(* CODESYS project 车床桁架_RECOVERED_2024-06-26T19-02-56.project
   CompiledLibraryCompatibilityVersion: LeadSysStudio V3.5 SP15 Patch 4
   Title: 车床桁架

Project tree, tasks and I/O mapping:
  Device : SC5-C0A4, Leadshine Technology Co., Ltd., order no. 504001, version 3.5.15.40
    application Application
      libraries: Standard, * (System); Util, * (System); CAA Net Base Services, 3.5.15.0 (CAA Technical Workgroup); HC_OmronUtils, 1.5.0.0 (Inovance); CmpHCUtils, 1.3.0.0 (Inovance); LS_IpoLib, 2.0.1.1 (Leadshine Technology Co.Ltd)
      task MainTask (cyclic, interval t#20ms, priority 1) calls PLC_PRG, Public_Prog, 信号, OP1002, OP1001, 回原, 气缸
      task EtherCAT_Master_Leadshine_A (cyclic, interval 4000 µs, priority 0) calls EtherCAT_Master_Leadshine_A.EtherCAT_Task, Servo_Ctrol
      program 回原 [LD]
      FunctionBlock/
        function block 点位范围判断 [ST]
        function block FB102_ClockPuls [LD]
        program Public_Prog [LD]: SystemVar
        function block FB_CylinderDouble [ST]
        function block FB_CylinderSingle [ST]
      global variables HMI
      global variables I_List
      global variables Alarm
      program POU [LD]
      Symbols
      data type CYLINDER_REF
      global variables 气缸_STRUCT
      program OP1002 [LD]: 辅助流程
      global variables System
      program 气缸 [LD]
      program Servo_Ctrol [LD]
      global variables Publics
      interface ITF
      global variables PersistentVars
      program 信号 [LD]
      program PLC_PRG [LD]
      program OP1001 [LD]
      global variables O_Lisk
    Device Diagnose
    Network Configuration
      LocalBus Config
    Resource Usage
    LocalBus_Master_Module : LocalBusR1 Master, Leadshine Technology Co., Ltd., version 3.5.15.40
      SC0032 : SC0032, Leadshine Technology Co., Ltd., version 3.5.15.40
          settings: 位置号 = 1
          unmapped channels: OUTPUT_0, OUTPUT_1, OUTPUT_2, OUTPUT_3
      SC3200 : SC3200, Leadshine Technology Co., Ltd., version 3.5.15.40
          settings: 位置号 = 0
          input  Application.I_List.X0 : BOOL  // INPUT_0.Bit0
          input  Application.I_List.X1 : BOOL  // INPUT_0.Bit1
          input  Application.I_List.X2 : BOOL  // INPUT_0.Bit2
          input  Application.I_List.X3 : BOOL  // INPUT_0.Bit3
          input  Application.I_List.X4 : BOOL  // INPUT_0.Bit4
          input  Application.I_List.X5 : BOOL  // INPUT_0.Bit5
          input  Application.I_List.X6 : BOOL  // INPUT_0.Bit6
          input  Application.I_List.X7 : BOOL  // INPUT_0.Bit7
          input  Application.I_List.X10 : BOOL  // INPUT_1.Bit0
          input  Application.I_List.X11 : BOOL  // INPUT_1.Bit1
          input  Application.I_List.X12 : BOOL  // INPUT_1.Bit2
          input  Application.I_List.X13 : BOOL  // INPUT_1.Bit3
          input  Application.I_List.X14 : BOOL  // INPUT_1.Bit4
          input  Application.I_List.X15 : BOOL  // INPUT_1.Bit5
          input  Application.I_List.X16 : BOOL  // INPUT_1.Bit6
          input  Application.I_List.X17 : BOOL  // INPUT_1.Bit7
          input  Application.I_List.X20 : BOOL  // INPUT_2.Bit0
          input  Application.I_List.X21 : BOOL  // INPUT_2.Bit1
          input  Application.I_List.X22 : BOOL  // INPUT_2.Bit2
          input  Application.I_List.X23 : BOOL  // INPUT_2.Bit3
          input  Application.I_List.X24 : BOOL  // INPUT_2.Bit4
          input  Application.I_List.X25 : BOOL  // INPUT_2.Bit5
          input  Application.I_List.X26 : BOOL  // INPUT_2.Bit6
          input  Application.I_List.X27 : BOOL  // INPUT_2.Bit7
          input  Application.I_List.X30 : BOOL  // INPUT_3.Bit0
          input  Application.I_List.X31 : BOOL  // INPUT_3.Bit1
          input  Application.I_List.X32 : BOOL  // INPUT_3.Bit2
          input  Application.I_List.X33 : BOOL  // INPUT_3.Bit3
          input  Application.I_List.X34 : BOOL  // INPUT_3.Bit4
          input  Application.I_List.X35 : BOOL  // INPUT_3.Bit5
          input  Application.I_List.X36 : BOOL  // INPUT_3.Bit6
          input  Application.I_List.X37 : BOOL  // INPUT_3.Bit7
          unmapped channels: INPUT_0, INPUT_1, INPUT_2, INPUT_3
    Modbus_Slave_RS232_COM : Modbus Slave RS232 COM, Leadshine Technology Co., Ltd., version 3.5.15.40
        settings: Vendor.Baudrate = 19200
    SoftMotion General Axis Pool
    ModbusTCP_Slave_Device : Modbus TCP Slave, Leadshine Technology Co., Ltd., version 00.00.00.10
    EtherCAT_Master_Leadshine_A : EtherCAT Master SoftMotion, 3S - Smart Software Solutions GmbH, version 3.5.16.30
        settings: NetworkName = 'ecat'; SelectNetworkByName = TRUE
      L6N_2 : L6N(COE), Leadshine Technology Co.,Ltd., order no. L6N, version Revision=16#00000001
          settings: DC sync0 cycletime = 4000; DC sync1 cycletime = 4000; Number of SDO = 6; Homing method.Index = 16#6098; Homing method.Subindex = 16#00; Homing method.Value = 19; Homing method.Size = 8; Homing method.AbortIfError = FALSE; Homing method.JumpToLine = FALSE; Homing method.Line = 0; Homing method.CompleteAccess = False; Homing velocity (fast).Index = 16#6099; Homing velocity (fast).Subindex = 16#01; Homing velocity (fast).Value = 3051735; Homing velocity (fast).Size = 32; Homing velocity (fast).AbortIfError = FALSE; Homing velocity (fast).JumpToLine = FALSE; Homing velocity (fast).Line = 0; Homing velocity (fast).CompleteAccess = False; Homing velocity (slow).Index = 16#6099; Homing velocity (slow).Subindex = 16#02; Homing velocity (slow).Value = 1220694; Homing velocity (slow).Size = 32; Homing velocity (slow).AbortIfError = FALSE; Homing velocity (slow).JumpToLine = FALSE; Homing velocity (slow).Line = 0; Homing velocity (slow).CompleteAccess = False; Homing acceleration.Index = 16#609A; Homing acceleration.Subindex = 16#00; Homing acceleration.Value = 61034692; Homing acceleration.Size = 32; Homing acceleration.AbortIfError = FALSE; Homing acceleration.JumpToLine = FALSE; Homing acceleration.Line = 0; Homing acceleration.CompleteAccess = False; Homing offset.Index = 16#607C; Homing offset.Subindex = 16#00; Homing offset.Value = 0; Homing offset.Size = 32; Homing offset.AbortIfError = FALSE;
            Homing offset.JumpToLine = FALSE; Homing offset.Line = 0; Homing offset.CompleteAccess = False
          unmapped channels: Control word, Profile target position, Touch Probe Function, Last error code, Status word, Modes of operation display, Position loop error, Actual motor torque, Actual motor position, Touch Probe Status, Touch probe pos1 pos value, Digital inputs
        Axis_2 : Axis, 3S - Smart Software Solutions GmbH, order no. 0, version 4.6.1.0
            settings: wDriveID = 2; dwRatioTechUnitsDenom = 524288000; iRatioTechUnitsNum = -859; fSWMaxVelocity = 687; fSWMaxAcceleration = 10000; fSWMaxDeceleration = 10000; fSWMaxJerk = 100000; 一圈脉冲数 = 8388608; 工作台一圈的位移 = 2; 电子齿轮比分子 = 100; 电子齿轮比分母 = 1; Commisioning.smci.Jerk = 0; ScalingIncs = 8388608; InvertDirection = True; AdrOffset_8010 = 28; BitOffset_8010 = 0; BitLength_8010 = 16; Address_8010 = '%QW14'; Type_8010 = 'UINT'; AddressPointer_8010 = ADR(%QW14); AdrOffset_8020 = 32; BitOffset_8020 = 0; BitLength_8020 = 32; Address_8020 = '%QD8'; Type_8020 = 'DINT'; AddressPointer_8020 = ADR(%QD8); AdrOffset_8030 = 4294967295; BitOffset_8030 = 0; BitLength_8030 = 32; Address_8030 = ''; Type_8030 = 'DINT'; AddressPointer_8030 = 0; AdrOffset_8040 = 4294967295; BitOffset_8040 = 0; BitLength_8040 = 16; Address_8040 = ''; Type_8040 = 'INT'; AddressPointer_8040 = 0; AdrOffset_8050 = 4294967295; BitOffset_8050 = 0;
              BitLength_8050 = 8; Address_8050 = ''; Type_8050 = 'SINT'; AddressPointer_8050 = 0; AdrOffset_8060 = 36; BitOffset_8060 = 0; BitLength_8060 = 16; Address_8060 = '%QW18'; Type_8060 = 'UINT'; AddressPointer_8060 = ADR(%QW18); AdrOffset_8070 = 4294967295; BitOffset_8070 = 0; BitLength_8070 = 0; Address_8070 = ''; Type_8070 = ''; AddressPointer_8070 = 0; AdrOffset_8080 = 4294967295; BitOffset_8080 = 0; BitLength_8080 = 16; Address_8080 = ''; Type_8080 = 'INT'; AddressPointer_8080 = 0; AdrOffset_8090 = 4294967295; BitOffset_8090 = 0; BitLength_8090 = 0; Address_8090 = ''; Type_8090 = ''; AddressPointer_8090 = 0; AdrOffset_8510 = 70; BitOffset_8510 = 0; BitLength_8510 = 16; Address_8510 = '%IW35'; Type_8510 = 'UINT'; AddressPointer_8510 = ADR(%IW35); AdrOffset_8520 = 84; BitOffset_8520 = 0; BitLength_8520 = 32; Address_8520 = '%ID21'; Type_8520 = 'DINT'; AddressPointer_8520 = ADR(%ID21);
              AdrOffset_8530 = 4294967295; BitOffset_8530 = 0; BitLength_8530 = 0; Address_8530 = ''; Type_8530 = ''; AddressPointer_8530 = 0; AdrOffset_8540 = 80; BitOffset_8540 = 0; BitLength_8540 = 16; Address_8540 = '%IW40'; Type_8540 = 'INT'; AddressPointer_8540 = ADR(%IW40); AdrOffset_8550 = 72; BitOffset_8550 = 0; BitLength_8550 = 8; Address_8550 = '%IB72'; Type_8550 = 'SINT'; AddressPointer_8550 = ADR(%IB72); AdrOffset_8560 = 96; BitOffset_8560 = 0; BitLength_8560 = 32; Address_8560 = '%ID24'; Type_8560 = 'UDINT'; AddressPointer_8560 = ADR(%ID24); AdrOffset_8570 = 88; BitOffset_8570 = 0; BitLength_8570 = 16; Address_8570 = '%IW44'; Type_8570 = 'UINT'; AddressPointer_8570 = ADR(%IW44); AdrOffset_8580 = 92; BitOffset_8580 = 0; BitLength_8580 = 32; Address_8580 = '%ID23'; Type_8580 = 'DINT'; AddressPointer_8580 = ADR(%ID23); AdrOffset_8590 = 4294967295; BitOffset_8590 = 0; BitLength_8590 = 0; Address_8590 = '';
              Type_8590 = ''; AddressPointer_8590 = 0; AdrOffset_8600 = 4294967295; BitOffset_8600 = 0; BitLength_8600 = 0; Address_8600 = ''; Type_8600 = ''; AddressPointer_8600 = 0; AdrOffset_8600 = 4294967295; BitOffset_8600 = 0; BitLength_8600 = 0; Address_8610 = ''; Type_8610 = ''; AddressPointer_8610 = 0; AdrOffset_8620 = 76; BitOffset_8620 = 0; BitLength_8620 = 32; Address_8620 = '%ID19'; Type_8620 = 'DINT'; AddressPointer_8620 = ADR(%ID19)
      L6N_1 : L6N(COE), Leadshine Technology Co.,Ltd., order no. L6N, version Revision=16#00000001
          settings: DC sync0 cycletime = 4000; DC sync1 cycletime = 4000; Number of SDO = 6; Homing method.Index = 16#6098; Homing method.Subindex = 16#00; Homing method.Value = 19; Homing method.Size = 8; Homing method.AbortIfError = FALSE; Homing method.JumpToLine = FALSE; Homing method.Line = 0; Homing method.CompleteAccess = FALSE; Homing velocity (fast).Index = 16#6099; Homing velocity (fast).Subindex = 16#01; Homing velocity (fast).Value = 8388608; Homing velocity (fast).Size = 32; Homing velocity (fast).AbortIfError = FALSE; Homing velocity (fast).JumpToLine = FALSE; Homing velocity (fast).Line = 0; Homing velocity (fast).CompleteAccess = FALSE; Homing velocity (slow).Index = 16#6099; Homing velocity (slow).Subindex = 16#02; Homing velocity (slow).Value = 3355443; Homing velocity (slow).Size = 32; Homing velocity (slow).AbortIfError = FALSE; Homing velocity (slow).JumpToLine = FALSE; Homing velocity (slow).Line = 0; Homing velocity (slow).CompleteAccess = FALSE; Homing acceleration.Index = 16#609A; Homing acceleration.Subindex = 16#00; Homing acceleration.Value = 167772160; Homing acceleration.Size = 32; Homing acceleration.AbortIfError = FALSE; Homing acceleration.JumpToLine = FALSE; Homing acceleration.Line = 0; Homing acceleration.CompleteAccess = FALSE; Homing offset.Index = 16#607C; Homing offset.Subindex = 16#00; Homing offset.Value = 0; Homing offset.Size = 32; Homing offset.AbortIfError = FALSE;
            Homing offset.JumpToLine = FALSE; Homing offset.Line = 0; Homing offset.CompleteAccess = FALSE
          unmapped channels: Control word, Profile target position, Touch Probe Function, Last error code, Status word, Modes of operation display, Position loop error, Actual motor torque, Actual motor position, Touch Probe Status, Touch probe pos1 pos value, Digital inputs
        Axis_1 : Axis, 3S - Smart Software Solutions GmbH, order no. 0, version 4.6.1.0
            settings: dwRatioTechUnitsDenom = 8388608; iRatioTechUnitsNum = -5; fSWMaxVelocity = 250; fSWMaxAcceleration = 1000; fSWMaxDeceleration = 10000; fSWMaxJerk = 100000; 一圈脉冲数 = 8388608; 工作台一圈的位移 = 5; 电子齿轮比分子 = 10; 电子齿轮比分母 = 100; ScalingIncs = 8388608; InvertDirection = True; AdrOffset_8010 = 16; BitOffset_8010 = 0; BitLength_8010 = 16; Address_8010 = '%QW8'; Type_8010 = 'UINT'; AddressPointer_8010 = ADR(%QW8); AdrOffset_8020 = 20; BitOffset_8020 = 0; BitLength_8020 = 32; Address_8020 = '%QD5'; Type_8020 = 'DINT'; AddressPointer_8020 = ADR(%QD5); AdrOffset_8030 = 4294967295; BitOffset_8030 = 0; BitLength_8030 = 32; Address_8030 = ''; Type_8030 = 'DINT'; AddressPointer_8030 = 0; AdrOffset_8040 = 4294967295; BitOffset_8040 = 0; BitLength_8040 = 16; Address_8040 = ''; Type_8040 = 'INT'; AddressPointer_8040 = 0; AdrOffset_8050 = 4294967295; BitOffset_8050 = 0; BitLength_8050 = 8; Address_8050 = '';
              Type_8050 = 'SINT'; AddressPointer_8050 = 0; AdrOffset_8060 = 24; BitOffset_8060 = 0; BitLength_8060 = 16; Address_8060 = '%QW12'; Type_8060 = 'UINT'; AddressPointer_8060 = ADR(%QW12); AdrOffset_8070 = 4294967295; BitOffset_8070 = 0; BitLength_8070 = 0; Address_8070 = ''; Type_8070 = ''; AddressPointer_8070 = 0; AdrOffset_8080 = 4294967295; BitOffset_8080 = 0; BitLength_8080 = 16; Address_8080 = ''; Type_8080 = 'INT'; AddressPointer_8080 = 0; AdrOffset_8090 = 4294967295; BitOffset_8090 = 0; BitLength_8090 = 0; Address_8090 = ''; Type_8090 = ''; AddressPointer_8090 = 0; AdrOffset_8510 = 38; BitOffset_8510 = 0; BitLength_8510 = 16; Address_8510 = '%IW19'; Type_8510 = 'UINT'; AddressPointer_8510 = ADR(%IW19); AdrOffset_8520 = 52; BitOffset_8520 = 0; BitLength_8520 = 32; Address_8520 = '%ID13'; Type_8520 = 'DINT'; AddressPointer_8520 = ADR(%ID13); AdrOffset_8530 = 4294967295; BitOffset_8530 = 0;
              BitLength_8530 = 0; Address_8530 = ''; Type_8530 = ''; AddressPointer_8530 = 0; AdrOffset_8540 = 48; BitOffset_8540 = 0; BitLength_8540 = 16; Address_8540 = '%IW24'; Type_8540 = 'INT'; AddressPointer_8540 = ADR(%IW24); AdrOffset_8550 = 40; BitOffset_8550 = 0; BitLength_8550 = 8; Address_8550 = '%IB40'; Type_8550 = 'SINT'; AddressPointer_8550 = ADR(%IB40); AdrOffset_8560 = 64; BitOffset_8560 = 0; BitLength_8560 = 32; Address_8560 = '%ID16'; Type_8560 = 'UDINT'; AddressPointer_8560 = ADR(%ID16); AdrOffset_8570 = 56; BitOffset_8570 = 0; BitLength_8570 = 16; Address_8570 = '%IW28'; Type_8570 = 'UINT'; AddressPointer_8570 = ADR(%IW28); AdrOffset_8580 = 60; BitOffset_8580 = 0; BitLength_8580 = 32; Address_8580 = '%ID15'; Type_8580 = 'DINT'; AddressPointer_8580 = ADR(%ID15); AdrOffset_8590 = 4294967295; BitOffset_8590 = 0; BitLength_8590 = 0; Address_8590 = ''; Type_8590 = ''; AddressPointer_8590 = 0;
              AdrOffset_8600 = 4294967295; BitOffset_8600 = 0; BitLength_8600 = 0; Address_8600 = ''; Type_8600 = ''; AddressPointer_8600 = 0; AdrOffset_8600 = 4294967295; BitOffset_8600 = 0; BitLength_8600 = 0; Address_8610 = ''; Type_8610 = ''; AddressPointer_8610 = 0; AdrOffset_8620 = 44; BitOffset_8620 = 0; BitLength_8620 = 32; Address_8620 = '%ID11'; Type_8620 = 'DINT'; AddressPointer_8620 = ADR(%ID11)
      L6N : L6N(COE), Leadshine Technology Co.,Ltd., order no. L6N, version Revision=16#00000001
          settings: DC sync0 cycletime = 4000; DC enable = 1; DC sync0 enable = 1; DC sync0 shift time = 0; DC sync1 cycletime = 4000; DC sync1 enable = 0; DC sync1 factor = 'x 1'; DC sync1 shift time = 0; Number of SDO = 6; Homing method.Index = 16#6098; Homing method.Subindex = 16#00; Homing method.Value = 19; Homing method.Size = 8; Homing method.AbortIfError = FALSE; Homing method.JumpToLine = FALSE; Homing method.Line = 0; Homing method.CompleteAccess = FALSE; Homing velocity (fast).Index = 16#6099; Homing velocity (fast).Subindex = 16#01; Homing velocity (fast).Value = 20971520; Homing velocity (fast).Size = 32; Homing velocity (fast).AbortIfError = FALSE; Homing velocity (fast).JumpToLine = FALSE; Homing velocity (fast).Line = 0; Homing velocity (fast).CompleteAccess = FALSE; Homing velocity (slow).Index = 16#6099; Homing velocity (slow).Subindex = 16#02; Homing velocity (slow).Value = 4194304; Homing velocity (slow).Size = 32; Homing velocity (slow).AbortIfError = FALSE; Homing velocity (slow).JumpToLine = FALSE; Homing velocity (slow).Line = 0; Homing velocity (slow).CompleteAccess = FALSE; Homing acceleration.Index = 16#609A; Homing acceleration.Subindex = 16#00; Homing acceleration.Value = 209715200; Homing acceleration.Size = 32; Homing acceleration.AbortIfError = FALSE; Homing acceleration.JumpToLine = FALSE; Homing acceleration.Line = 0;
            Homing acceleration.CompleteAccess = FALSE; Homing offset.Index = 16#607C; Homing offset.Subindex = 16#00; Homing offset.Value = 0; Homing offset.Size = 32; Homing offset.AbortIfError = FALSE; Homing offset.JumpToLine = FALSE; Homing offset.Line = 0; Homing offset.CompleteAccess = FALSE
          unmapped channels: Control word, Profile target position, Touch Probe Function, Last error code, Status word, Modes of operation display, Position loop error, Actual motor torque, Actual motor position, Touch Probe Status, Touch probe pos1 pos value, Digital inputs
        Axis : Axis, 3S - Smart Software Solutions GmbH, order no. 0, version 4.6.1.0
            settings: wDriveID = 0; dwRatioTechUnitsDenom = 2097152; iRatioTechUnitsNum = -1; fSWMaxVelocity = 200; fSWMaxAcceleration = 1000; fSWMaxDeceleration = 10000; fSWMaxJerk = 100000; 一圈脉冲数 = 10; 工作台一圈的位移 = 20; 电子齿轮比分子 = 100; 电子齿轮比分母 = 100; ScalingIncs = 8388608; InvertDirection = True; AdrOffset_8010 = 4; BitOffset_8010 = 0; BitLength_8010 = 16; Address_8010 = '%QW2'; Type_8010 = 'UINT'; AddressPointer_8010 = ADR(%QW2); AdrOffset_8020 = 8; BitOffset_8020 = 0; BitLength_8020 = 32; Address_8020 = '%QD2'; Type_8020 = 'DINT'; AddressPointer_8020 = ADR(%QD2); AdrOffset_8030 = 4294967295; BitOffset_8030 = 0; BitLength_8030 = 32; Address_8030 = ''; Type_8030 = 'DINT'; AddressPointer_8030 = 0; AdrOffset_8040 = 4294967295; BitOffset_8040 = 0; BitLength_8040 = 16; Address_8040 = ''; Type_8040 = 'INT'; AddressPointer_8040 = 0; AdrOffset_8050 = 4294967295; BitOffset_8050 = 0; BitLength_8050 = 8;
              Address_8050 = ''; Type_8050 = 'SINT'; AddressPointer_8050 = 0; AdrOffset_8060 = 12; BitOffset_8060 = 0; BitLength_8060 = 16; Address_8060 = '%QW6'; Type_8060 = 'UINT'; AddressPointer_8060 = ADR(%QW6); AdrOffset_8070 = 4294967295; BitOffset_8070 = 0; BitLength_8070 = 0; Address_8070 = ''; Type_8070 = ''; AddressPointer_8070 = 0; AdrOffset_8080 = 4294967295; BitOffset_8080 = 0; BitLength_8080 = 16; Address_8080 = ''; Type_8080 = 'INT'; AddressPointer_8080 = 0; AdrOffset_8090 = 4294967295; BitOffset_8090 = 0; BitLength_8090 = 0; Address_8090 = ''; Type_8090 = ''; AddressPointer_8090 = 0; AdrOffset_8510 = 6; BitOffset_8510 = 0; BitLength_8510 = 16; Address_8510 = '%IW3'; Type_8510 = 'UINT'; AddressPointer_8510 = ADR(%IW3); AdrOffset_8520 = 20; BitOffset_8520 = 0; BitLength_8520 = 32; Address_8520 = '%ID5'; Type_8520 = 'DINT'; AddressPointer_8520 = ADR(%ID5); AdrOffset_8530 = 4294967295;
              BitOffset_8530 = 0; BitLength_8530 = 0; Address_8530 = ''; Type_8530 = ''; AddressPointer_8530 = 0; AdrOffset_8540 = 16; BitOffset_8540 = 0; BitLength_8540 = 16; Address_8540 = '%IW8'; Type_8540 = 'INT'; AddressPointer_8540 = ADR(%IW8); AdrOffset_8550 = 8; BitOffset_8550 = 0; BitLength_8550 = 8; Address_8550 = '%IB8'; Type_8550 = 'SINT'; AddressPointer_8550 = ADR(%IB8); AdrOffset_8560 = 32; BitOffset_8560 = 0; BitLength_8560 = 32; Address_8560 = '%ID8'; Type_8560 = 'UDINT'; AddressPointer_8560 = ADR(%ID8); AdrOffset_8570 = 24; BitOffset_8570 = 0; BitLength_8570 = 16; Address_8570 = '%IW12'; Type_8570 = 'UINT'; AddressPointer_8570 = ADR(%IW12); AdrOffset_8580 = 28; BitOffset_8580 = 0; BitLength_8580 = 32; Address_8580 = '%ID7'; Type_8580 = 'DINT'; AddressPointer_8580 = ADR(%ID7); AdrOffset_8590 = 4294967295; BitOffset_8590 = 0; BitLength_8590 = 0; Address_8590 = ''; Type_8590 = '';
              AddressPointer_8590 = 0; AdrOffset_8600 = 4294967295; BitOffset_8600 = 0; BitLength_8600 = 0; Address_8600 = ''; Type_8600 = ''; AddressPointer_8600 = 0; AdrOffset_8600 = 4294967295; BitOffset_8600 = 0; BitLength_8600 = 0; Address_8610 = ''; Type_8610 = ''; AddressPointer_8610 = 0; AdrOffset_8620 = 12; BitOffset_8620 = 0; BitLength_8620 = 32; Address_8620 = '%ID3'; Type_8620 = 'DINT'; AddressPointer_8620 = ADR(%ID3)
      L6N_3 : L6N(COE), Leadshine Technology Co.,Ltd., order no. L6N, version Revision=16#00000001
          settings: DC sync0 cycletime = 4000; DC sync1 cycletime = 4000; Number of SDO = 6; Homing method.Index = 16#6098; Homing method.Subindex = 16#00; Homing method.Value = 29; Homing method.Size = 8; Homing method.AbortIfError = FALSE; Homing method.JumpToLine = FALSE; Homing method.Line = 0; Homing method.CompleteAccess = False; Homing velocity (fast).Index = 16#6099; Homing velocity (fast).Subindex = 16#01; Homing velocity (fast).Value = 3051735; Homing velocity (fast).Size = 32; Homing velocity (fast).AbortIfError = FALSE; Homing velocity (fast).JumpToLine = FALSE; Homing velocity (fast).Line = 0; Homing velocity (fast).CompleteAccess = False; Homing velocity (slow).Index = 16#6099; Homing velocity (slow).Subindex = 16#02; Homing velocity (slow).Value = 1220694; Homing velocity (slow).Size = 32; Homing velocity (slow).AbortIfError = FALSE; Homing velocity (slow).JumpToLine = FALSE; Homing velocity (slow).Line = 0; Homing velocity (slow).CompleteAccess = False; Homing acceleration.Index = 16#609A; Homing acceleration.Subindex = 16#00; Homing acceleration.Value = 61034692; Homing acceleration.Size = 32; Homing acceleration.AbortIfError = FALSE; Homing acceleration.JumpToLine = FALSE; Homing acceleration.Line = 0; Homing acceleration.CompleteAccess = False; Homing offset.Index = 16#607C; Homing offset.Subindex = 16#00; Homing offset.Value = 0; Homing offset.Size = 32; Homing offset.AbortIfError = FALSE;
            Homing offset.JumpToLine = FALSE; Homing offset.Line = 0; Homing offset.CompleteAccess = False
          unmapped channels: Control word, Profile target position, Touch Probe Function, Last error code, Status word, Modes of operation display, Position loop error, Actual motor torque, Actual motor position, Touch Probe Status, Touch probe pos1 pos value, Digital inputs
        Axis_3 : Axis, 3S - Smart Software Solutions GmbH, order no. 0, version 4.6.1.0
            settings: wDriveID = 3; dwRatioTechUnitsDenom = 3814564139; iRatioTechUnitsNum = 10000; fSWMaxVelocity = 1099; fSWMaxAcceleration = 1000; fSWMaxDeceleration = 10000; fSWMaxJerk = 100000; 一圈脉冲数 = 10; 工作台一圈的位移 = 20; 电子齿轮比分子 = 100; 电子齿轮比分母 = 100; ScalingIncs = 8388608; AdrOffset_8010 = 40; BitOffset_8010 = 0; BitLength_8010 = 16; Address_8010 = '%QW20'; Type_8010 = 'UINT'; AddressPointer_8010 = ADR(%QW20); AdrOffset_8020 = 44; BitOffset_8020 = 0; BitLength_8020 = 32; Address_8020 = '%QD11'; Type_8020 = 'DINT'; AddressPointer_8020 = ADR(%QD11); AdrOffset_8030 = 4294967295; BitOffset_8030 = 0; BitLength_8030 = 32; Address_8030 = ''; Type_8030 = 'DINT'; AddressPointer_8030 = 0; AdrOffset_8040 = 4294967295; BitOffset_8040 = 0; BitLength_8040 = 16; Address_8040 = ''; Type_8040 = 'INT'; AddressPointer_8040 = 0; AdrOffset_8050 = 4294967295; BitOffset_8050 = 0; BitLength_8050 = 8; Address_8050 = '';
              Type_8050 = 'SINT'; AddressPointer_8050 = 0; AdrOffset_8060 = 48; BitOffset_8060 = 0; BitLength_8060 = 16; Address_8060 = '%QW24'; Type_8060 = 'UINT'; AddressPointer_8060 = ADR(%QW24); AdrOffset_8070 = 4294967295; BitOffset_8070 = 0; BitLength_8070 = 0; Address_8070 = ''; Type_8070 = ''; AddressPointer_8070 = 0; AdrOffset_8080 = 4294967295; BitOffset_8080 = 0; BitLength_8080 = 16; Address_8080 = ''; Type_8080 = 'INT'; AddressPointer_8080 = 0; AdrOffset_8090 = 4294967295; BitOffset_8090 = 0; BitLength_8090 = 0; Address_8090 = ''; Type_8090 = ''; AddressPointer_8090 = 0; AdrOffset_8510 = 102; BitOffset_8510 = 0; BitLength_8510 = 16; Address_8510 = '%IW51'; Type_8510 = 'UINT'; AddressPointer_8510 = ADR(%IW51); AdrOffset_8520 = 116; BitOffset_8520 = 0; BitLength_8520 = 32; Address_8520 = '%ID29'; Type_8520 = 'DINT'; AddressPointer_8520 = ADR(%ID29); AdrOffset_8530 = 4294967295; BitOffset_8530 = 0;
              BitLength_8530 = 0; Address_8530 = ''; Type_8530 = ''; AddressPointer_8530 = 0; AdrOffset_8540 = 112; BitOffset_8540 = 0; BitLength_8540 = 16; Address_8540 = '%IW56'; Type_8540 = 'INT'; AddressPointer_8540 = ADR(%IW56); AdrOffset_8550 = 104; BitOffset_8550 = 0; BitLength_8550 = 8; Address_8550 = '%IB104'; Type_8550 = 'SINT'; AddressPointer_8550 = ADR(%IB104); AdrOffset_8560 = 128; BitOffset_8560 = 0; BitLength_8560 = 32; Address_8560 = '%ID32'; Type_8560 = 'UDINT'; AddressPointer_8560 = ADR(%ID32); AdrOffset_8570 = 120; BitOffset_8570 = 0; BitLength_8570 = 16; Address_8570 = '%IW60'; Type_8570 = 'UINT'; AddressPointer_8570 = ADR(%IW60); AdrOffset_8580 = 124; BitOffset_8580 = 0; BitLength_8580 = 32; Address_8580 = '%ID31'; Type_8580 = 'DINT'; AddressPointer_8580 = ADR(%ID31); AdrOffset_8590 = 4294967295; BitOffset_8590 = 0; BitLength_8590 = 0; Address_8590 = ''; Type_8590 = ''; AddressPointer_8590 = 0;
              AdrOffset_8600 = 4294967295; BitOffset_8600 = 0; BitLength_8600 = 0; Address_8600 = ''; Type_8600 = ''; AddressPointer_8600 = 0; AdrOffset_8600 = 4294967295; BitOffset_8600 = 0; BitLength_8600 = 0; Address_8610 = ''; Type_8610 = ''; AddressPointer_8610 = 0; AdrOffset_8620 = 108; BitOffset_8620 = 0; BitLength_8620 = 32; Address_8620 = '%ID27'; Type_8620 = 'DINT'; AddressPointer_8620 = ADR(%ID27)
*)

// Device/Application/CYLINDER_REF
TYPE CYLINDER_REF :
STRUCT
	///初始化时返回原位控制
	xInit: BOOL;
	///自动控制,变为TRUE时，执行到位控制，变为FALSE时执行原位控制
	xAutoCmd: BOOL;
	///到位标志,处于原位状态
	xIsBack: BOOL;
	///到位标志,处于到位状态	
	xIsFront: BOOL;
END_STRUCT
END_TYPE

// Device/Application/HMI
{attribute 'qualified_only'}
VAR_GLOBAL
END_VAR
VAR_GLOBAL
	报警复位 AT %MX0.0: BOOL;
END_VAR
VAR_GLOBAL RETAIN PERSISTENT
	上料推出气缸原位延时 AT %MW1002: WORD := 10;
	上料推出气缸到位延时 AT %MW1003: WORD := 10;
END_VAR
VAR_GLOBAL
	上料顶起气缸_ON_UP AT %MX0.3: BOOL;
END_VAR
VAR_GLOBAL RETAIN PERSISTENT
	上料顶起气缸原位延时 AT %MW1000: WORD := 10;
	上料顶起气缸到位位延时 AT %MW1001: WORD := 10;
END_VAR
VAR_GLOBAL
	上料气动振动筛_ON_UP AT %MX0.6: BOOL;
	X轴失能 AT %MX0.7: BOOL;
	Z2轴失能 AT %MX1.0: BOOL;
	Z1轴失能 AT %MX1.1: BOOL;
	Y轴失能 AT %MX1.2: BOOL;
	X轴_CCW AT %MX1.3: BOOL;
	X轴_CW AT %MX1.4: BOOL;
	Y轴_CCW AT %MX1.5: BOOL;
	Y轴_CW AT %MX0.5: BOOL;
	Z1轴_CCW AT %MX0.4: BOOL;
	Z1轴_CW AT %MX1.6: BOOL;
	Z2轴_CCW AT %MX0.2: BOOL;
	Z2轴_CW AT %MX0.1: BOOL;
	上料推出气缸_ON_UP AT %MX1.7: BOOL;
END_VAR
VAR_GLOBAL RETAIN PERSISTENT
	X轴手动速度 AT %MD1000: REAL := 20;
	Z1轴手动速度 AT %MD1002: REAL := 20;
	Y轴手动速度 AT %MD1001: REAL := 20;
	Z2轴手动速度 AT %MD1003: REAL := 20;
	X轴手动减速度: REAL := 1000;
	X轴手动加速度: REAL := 1000;
	Y轴手动加速度: REAL := 1000;
	Y轴手动减速度: REAL := 1000;
	Z1轴手动减速度: REAL := 1000;
	Z1轴手动加速度: REAL := 1000;
	Z2轴手动减速度: REAL := 1000;
	Z2轴手动加速度: REAL := 1000;
END_VAR
VAR_GLOBAL
	X轴错误代码 AT %MD30000: DWORD;
	X状态_未使能 AT %MX2.4: BOOL;
	X状态_报错 AT %MX2.5: BOOL;
	X状态_停止中 AT %MX2.6: BOOL;
	X状态_准备好 AT %MX2.7: BOOL;
	X状态_点位运动 AT %MX3.0: BOOL;
	X状态_连续运动: BOOL;
	X状态_同步运动: BOOL;
	X状态_回零中: BOOL;
	X状态_恒速运动 AT %MX3.1: BOOL;
	X状态_加速中 AT %MX3.2: BOOL;
	X状态_减速中 AT %MX3.3: BOOL;
	X状态_超过软限制 AT %MX3.4: BOOL;
	Y轴错误代码 AT %MD30001: DWORD;
	Y状态_未使能 AT %MX3.5: BOOL;
	Y状态_报错 AT %MX3.6: BOOL;
	Y状态_停止中 AT %MX3.7: BOOL;
	Y状态_准备好 AT %MX4.0: BOOL;
	Y状态_点位运动 AT %MX4.1: BOOL;
	Y状态_连续运动: BOOL;
	Y状态_同步运动: BOOL;
	Y状态_回零中: BOOL;
	Y状态_恒速运动 AT %MX4.2: BOOL;
	Y状态_加速中 AT %MX4.3: BOOL;
	Y状态_减速中 AT %MX4.4: BOOL;
	Y状态_超过软限制 AT %MX4.5: BOOL;
	Z1轴错误代码 AT %MD30002: DWORD;
	Z1状态_未使能 AT %MX4.6: BOOL;
	Z1状态_报错 AT %MX4.7: BOOL;
	Z1状态_停止中 AT %MX5.0: BOOL;
	Z1状态_准备好 AT %MX5.1: BOOL;
	Z1状态_点位运动 AT %MX5.2: BOOL;
	Z1状态_连续运动: BOOL;
	Z1状态_同步运动: BOOL;
	Z1状态_回零中: BOOL;
	Z1状态_恒速运动 AT %MX5.3: BOOL;
	Z1状态_加速中 AT %MX5.4: BOOL;
	Z1状态_减速中 AT %MX5.5: BOOL;
	Z1状态_超过软限制 AT %MX5.6: BOOL;
	Z2轴错误代码 AT %MD30003: DWORD;
	Z2状态_未使能 AT %MX5.7: BOOL;
	Z2状态_报错 AT %mx6.0: BOOL;
	Z2状态_停止中 AT %mx6.1: BOOL;
	Z2状态_准备好 AT %MX6.7: BOOL;
	Z2状态_点位运动 AT %MX6.2: BOOL;
	Z2状态_连续运动: BOOL;
	Z2状态_同步运动: BOOL;
	Z2状态_回零中: BOOL;
	Z2状态_恒速运动 AT %MX6.3: BOOL;
	Z2状态_加速中 AT %MX6.4: BOOL;
	Z2状态_减速中 AT %MX6.5: BOOL;
	Z2状态_超过软限制 AT %MX6.6: BOOL;
	上料气爪_ON_UP AT %MX2.3: BOOL;
	开门气缸_ON_UP AT %MX2.2: BOOL;
	翻转气缸_ON_UP AT %MX2.1: BOOL;
	下料气爪_ON_UP AT %MX2.0: BOOL;
END_VAR
VAR_GLOBAL RETAIN PERSISTENT
	点位P0 AT %MD2000: ARRAY[0..3] OF REAL;
	点位P1 AT %MD2004: ARRAY[0..3] OF REAL;
END_VAR

VAR_GLOBAL
	Y轴当前位置 AT %MD1005: REAL;
	Z2轴当前位置 AT %MD1007: REAL;
	Z1轴当前位置 AT %MD1006: REAL;
	X轴当前位置 AT %MD1004: REAL;
	Z2当前速度: REAL;
	Z1当前速度: REAL;
	Y轴当前速度: REAL;
	X轴当前速度: REAL;
END_VAR
VAR_GLOBAL RETAIN PERSISTENT
	上料气爪原位延时 AT %MW1004: WORD := 10;
	上料气爪到位延时 AT %MW1005: WORD := 10;
	下料气爪到位延时 AT %MW1006: WORD := 10;
	下料气爪原位延时 AT %MW1007: WORD := 10;
	翻转气爪到位延时 AT %MW1008: WORD := 10;
	翻转气爪原位延时 AT %MW1009: WORD := 10;
	开门气缸原位延时 AT %MW1010: WORD := 50;
	开门气缸到位延时 AT %MW1011: WORD := 50;
	点位P9 AT %MD2036: ARRAY[0..3] OF REAL;
	点位P8 AT %MD2032: ARRAY[0..3] OF REAL;
	点位P7 AT %MD2028: ARRAY[0..3] OF REAL;
	点位P6 AT %MD2024: ARRAY[0..3] OF REAL;
	点位P5 AT %MD2020: ARRAY[0..3] OF REAL;
	点位P4 AT %MD2016: ARRAY[0..3] OF REAL;
	点位P3 AT %MD2012: ARRAY[0..3] OF REAL;
	点位P2 AT %MD2008: ARRAY[0..3] OF REAL;
	点位P10 AT %MD2040: ARRAY[0..3] OF REAL;
END_VAR
VAR_GLOBAL
	Z2回零触发 AT %MX7.3: BOOL;
	Z1回零触发 AT %MX7.2: BOOL;
	Y回零触发 AT %MX7.1: BOOL;
	X回零触发 AT %MX7.0: BOOL;
	Y回零完成 AT %MX7.5: BOOL;
	Z2回零完成 AT %MX7.7: BOOL;
	Z1回零完成 AT %MX7.6: BOOL;
	X回零完成 AT %MX7.4: BOOL;
	空循环模式 AT %MX8.0: BOOL;
	排空模式 AT %MX8.1: BOOL;
	P1范围内 AT %MX8.2: BOOL;
	P2范围内 AT %MX8.3: BOOL;
	P3范围内 AT %MX8.4: BOOL;
	P4范围内 AT %MX8.5: BOOL;
	P5范围内 AT %MX8.6: BOOL;
	P6范围内 AT %MX8.7: BOOL;
	P7范围内 AT %MX9.0: BOOL;
	P8范围内 AT %MX9.1: BOOL;
	P9范围内 AT %MX9.2: BOOL;
	P10范围内 AT %MX9.3: BOOL;
END_VAR
VAR_GLOBAL RETAIN PERSISTENT
	点位P12 AT %MD2048: ARRAY[0..3] OF REAL;
	点位P11 AT %MD2044: ARRAY[0..3] OF REAL;
	点位P13 AT %MD2052: ARRAY[0..3] OF REAL;
	点位P14 AT %MD2056: ARRAY[0..3] OF REAL;
END_VAR
VAR_GLOBAL
	原点状态 AT %MW1012: WORD := 0;
	设备回原触发 AT %MX9.4: BOOL;
	设备状态 AT %MW1013: WORD;
END_VAR
VAR_GLOBAL RETAIN PERSISTENT
	X最大速度 AT %MD1010: REAL := 100;
	Y最大速度 AT %MD1011: REAL := 100;
	Z1最大速度 AT %MD1012: REAL := 100;
	Z2最大速度 AT %MD1013: REAL := 100;
	X速度比例 AT %MD1014: REAL := 10;
	Y速度比例 AT %MD1015: REAL := 10;
	Z1速度比例 AT %MD1016: REAL := 10;
	Z2速度比例 AT %MD1017: REAL := 10;
END_VAR

// Device/Application/I_List
{attribute 'qualified_only'}
VAR_GLOBAL
	// 上料传送带到位确认
	X0: BOOL;
	// 紧急停止
	X1: BOOL;
	// 推出气缸原位
	X2: BOOL;
	// 推出气缸动作位
	X3: BOOL;
	// 顶起气缸原位
	X4: BOOL;
	// 顶起气缸动作位
	X5: BOOL;
	// 上料气爪原位
	X6: BOOL;
	// 上料气爪动作位
	X7: BOOL;
	// 下料气爪原位
	X10: BOOL;
	// 下料气爪动作位
	X11: BOOL;
	// 翻转气缸原位
	X12: BOOL;
	// 翻转气缸动作位
	X13: BOOL;
	// 开门气缸原位
	X14: BOOL;
	// 开门气缸动作位
	X15: BOOL;
	// 启动按钮
	X16: BOOL;
	// 停止按钮
	X17: BOOL;
	// 复位按钮
	X20: BOOL;
	// 手自动按钮ON为自动
	X21: BOOL;
	// 下料确认
	X22: BOOL;
	// 联机卡盘夹紧
	X23: BOOL;
	// 联机启动
	X24: BOOL;
	// 联机停止
	X25: BOOL;
	// 联机故障
	X26: BOOL;
	// 联机X轴零点
	X27: BOOL;
	// 联机Z轴零点
	X30: BOOL;
	// 门
	X31: BOOL;
	// 门
	X32: BOOL;
	// 油泵报警
	X33: BOOL;
	X34: BOOL;
	X35: BOOL;
	X36: BOOL;
	X37: BOOL;
END_VAR

// Device/Application/Alarm
{attribute 'qualified_only'}
VAR_GLOBAL
END_VAR
VAR_GLOBAL
	设备急停 AT %MX100.0: BOOL;
	推出气缸手自动不一致报警 AT %MX100.1: BOOL;
	推出气缸原位报警 AT %MX100.2: BOOL;
	推出气缸到位报警 AT %MX100.3: BOOL;
	顶起气缸手自动不一致报警 AT %MX100.4: BOOL;
	顶起气缸原位报警 AT %MX100.5: BOOL;
	顶起气缸到位报警 AT %MX100.6: BOOL;
	上料气爪手自动不一致报警 AT %MX100.7: BOOL;
	上料气爪原位报警 AT %MX101.0: BOOL;
	上料气爪到位报警 AT %MX101.1: BOOL;
	下料气爪手自动不一致报警 AT %MX101.2: BOOL;
	下料气爪原位报警 AT %MX101.3: BOOL;
	下料气爪到位报警 AT %MX101.4: BOOL;
	翻转气缸手自动不一致报警 AT %MX101.5: BOOL;
	翻转气缸原位报警 AT %MX101.6: BOOL;
	翻转气缸到位报警 AT %MX101.7: BOOL;
	开门气缸手自动不一致报警 AT %MX102.0: BOOL;
	开门气缸原位报警 AT %MX102.1: BOOL;
	开门气缸到位报警 AT %MX102.2: BOOL;
END_VAR

// Device/Application/气缸_STRUCT
{attribute 'qualified_only'}
VAR_GLOBAL
	上料推出气缸: CYLINDER_REF;
	上料顶起气缸: CYLINDER_REF;
	上料振动筛: CYLINDER_REF;
	开门气缸: CYLINDER_REF;
	翻转气缸: CYLINDER_REF;
	上料气爪: CYLINDER_REF;
	下料气爪: CYLINDER_REF;
END_VAR

// Device/Application/System
{attribute 'qualified_only'}
VAR_GLOBAL
	// 上电扫描一周期
FirstScan    :BOOL;
// 常ON
AlwaysTRUE   : BOOL;
// 常OFF
AlwaysFALSE  : BOOL;
// 0.1S周期脉冲
Clock_10Hz    :BOOL;
// 0.2S周期脉冲
Clock_5Hz    :BOOL;
// 0.5S周期脉冲
Clock_2Hz    :BOOL;
// 1S周期脉冲
Clock_1Hz    :BOOL;
// 2S周期脉冲
Clock_HalfHz :BOOL;
END_VAR

// Device/Application/Publics
{attribute 'qualified_only'}
VAR_GLOBAL
	// 调试使用常ON
CYGIA_ON   :BOOL;
// 调试使用常OFF
CYGIA_OFF  :BOOL;
	启动上升: BOOL;
	警报: BOOL;
	暂停: BOOL;
	EMG: BOOL;
	X定位数据: REAL;
	Y定位数据: REAL;
	Z1定位数据: REAL;
	Z2定位数据: REAL;
END_VAR
VAR_GLOBAL RETAIN PERSISTENT
	Z2加速度 AT %MD1083: REAL;
	Z1加速度 AT %MD1082: REAL;
	Y加速度 AT %MD1081: REAL;
	X加速度 AT %MD1080: REAL;
	Z2减速度 AT %MD1087: REAL;
	Z1减速度 AT %MD1086: REAL;
	Y减速度 AT %MD1085: REAL;
	X减速度 AT %MD1084: REAL;
	Z2自动速度: REAL;
	Z1自动速度: REAL;
	Y自动速度: REAL;
	X自动速度: REAL;
END_VAR
VAR_GLOBAL
	Z2轴完成: BOOL;
	Z1轴完成: BOOL;
	Y轴完成: BOOL;
	X轴完成: BOOL;
	Z2轴启动: BOOL;
	Z1轴启动: BOOL;
	Y轴启动: BOOL;
	X轴启动: BOOL;
END_VAR

// Device/Application/PersistentVars
{attribute 'qualified_only'}
VAR_GLOBAL PERSISTENT RETAIN
	// 生成持久变量的实例路径
	HMI.上料推出气缸原位延时: WORD := WORD#10;
	// 生成持久变量的实例路径
	HMI.上料推出气缸到位延时: WORD := WORD#10;
	// 生成持久变量的实例路径
	HMI.上料顶起气缸原位延时: WORD := WORD#10;
	// 生成持久变量的实例路径
	HMI.上料顶起气缸到位位延时: WORD := WORD#10;
	// 生成持久变量的实例路径
	HMI.X轴手动速度: REAL := 20.0;
	// 生成持久变量的实例路径
	HMI.Z1轴手动速度: REAL := 20.0;
	// 生成持久变量的实例路径
	HMI.Y轴手动速度: REAL := 20.0;
	// 生成持久变量的实例路径
	HMI.Z2轴手动速度: REAL := 20.0;
	// 生成持久变量的实例路径
	HMI.X轴手动减速度: REAL := 1000.0;
	// 生成持久变量的实例路径
	HMI.X轴手动加速度: REAL := 1000.0;
	// 生成持久变量的实例路径
	HMI.Y轴手动加速度: REAL := 1000.0;
	// 生成持久变量的实例路径
	HMI.Y轴手动减速度: REAL := 1000.0;
	// 生成持久变量的实例路径
	HMI.Z1轴手动减速度: REAL := 1000.0;
	// 生成持久变量的实例路径
	HMI.Z1轴手动加速度: REAL := 1000.0;
	// 生成持久变量的实例路径
	HMI.Z2轴手动减速度: REAL := 1000.0;
	// 生成持久变量的实例路径
	HMI.Z2轴手动加速度: REAL := 1000.0;
	// 生成持久变量的实例路径
	HMI.点位P1: ARRAY [0..3] OF REAL;
	// 生成持久变量的实例路径
	HMI.点位P0: ARRAY [0..3] OF REAL;
	// 生成持久变量的实例路径
	HMI.点位P9: ARRAY [0..3] OF REAL;
	// 生成持久变量的实例路径
	HMI.点位P8: ARRAY [0..3] OF REAL;
	// 生成持久变量的实例路径
	HMI.点位P7: ARRAY [0..3] OF REAL;
	// 生成持久变量的实例路径
	HMI.点位P6: ARRAY [0..3] OF REAL;
	// 生成持久变量的实例路径
	HMI.点位P5: ARRAY [0..3] OF REAL;
	// 生成持久变量的实例路径
	HMI.点位P4: ARRAY [0..3] OF REAL;
	// 生成持久变量的实例路径
	HMI.点位P3: ARRAY [0..3] OF REAL;
	// 生成持久变量的实例路径
	HMI.点位P2: ARRAY [0..3] OF REAL;
	// 生成持久变量的实例路径
	HMI.点位P10: ARRAY [0..3] OF REAL;
	// 生成持久变量的实例路径
	HMI.上料气爪原位延时: WORD := WORD#10;
	// 生成持久变量的实例路径
	HMI.上料气爪到位延时: WORD := WORD#10;
	// 生成持久变量的实例路径
	HMI.下料气爪到位延时: WORD := WORD#10;
	// 生成持久变量的实例路径
	HMI.下料气爪原位延时: WORD := WORD#10;
	// 生成持久变量的实例路径
	HMI.翻转气爪到位延时: WORD := WORD#10;
	// 生成持久变量的实例路径
	HMI.翻转气爪原位延时: WORD := WORD#10;
	// 生成持久变量的实例路径
	HMI.开门气缸原位延时: WORD := 50;
	// 生成持久变量的实例路径
	HMI.开门气缸到位延时: WORD := 50;
	// 生成持久变量的实例路径
	Publics.Y加速度: REAL;
	// 生成持久变量的实例路径
	Publics.X加速度: REAL;
	// 生成持久变量的实例路径
	Publics.Z2减速度: REAL;
	// 生成持久变量的实例路径
	Publics.Z1减速度: REAL;
	// 生成持久变量的实例路径
	Publics.Y减速度: REAL;
	// 生成持久变量的实例路径
	Publics.X减速度: REAL;
	// 生成持久变量的实例路径
	Publics.Z2自动速度: REAL;
	// 生成持久变量的实例路径
	Publics.Z1自动速度: REAL;
	// 生成持久变量的实例路径
	Publics.Y自动速度: REAL;
	// 生成持久变量的实例路径
	Publics.X自动速度: REAL;
	// 生成持久变量的实例路径
	HMI.点位P12: ARRAY [0..3] OF REAL;
	// 生成持久变量的实例路径
	HMI.点位P11: ARRAY [0..3] OF REAL;
	// 生成持久变量的实例路径
	HMI.点位P13: ARRAY [0..3] OF REAL;
	// 生成持久变量的实例路径
	HMI.点位P14: ARRAY [0..3] OF REAL;
	// 生成持久变量的实例路径
	HMI.X最大速度: REAL := 100.0;
	// 生成持久变量的实例路径
	HMI.Y最大速度: REAL := 100.0;
	// 生成持久变量的实例路径
	HMI.Z1最大速度: REAL := 100.0;
	// 生成持久变量的实例路径
	HMI.Z2最大速度: REAL := 100.0;
	// 生成持久变量的实例路径
	HMI.X速度比例: REAL := 10.0;
	// 生成持久变量的实例路径
	HMI.Y速度比例: REAL := 10.0;
	// 生成持久变量的实例路径
	HMI.Z1速度比例: REAL := 10.0;
	// 生成持久变量的实例路径
	HMI.Z2速度比例: REAL := 10.0;
	// 生成持久变量的实例路径
	Publics.Z2加速度: REAL;
	// 生成持久变量的实例路径
	Publics.Z1加速度: REAL;
END_VAR

// Device/Application/O_Lisk
{attribute 'qualified_only'}
VAR_GLOBAL
	// 皮带运转
	Y0 AT %QX0.0: BOOL;
	// 震动筛运动
	Y1 AT %QX0.1: BOOL;
	// 推出气缸原位
	Y2 AT %QX0.2: BOOL;
	// 紧急停止输出
	Y3 AT %QX0.3: BOOL;
	// 顶起气缸原位
	Y4 AT %QX0.4: BOOL;
	Y5 AT %QX0.5: BOOL;
	// 上料气爪原位
	Y6 AT %QX0.6: BOOL;
	Y7 AT %QX0.7: BOOL;
	// 下料气爪原位
	Y10 AT %QX1.0: BOOL;
	Y11 AT %QX1.1: BOOL;
	// 翻转气缸原位
	Y12 AT %QX1.2: BOOL;
	Y13 AT %QX1.3: BOOL;
	// 开门气缸原位
	Y14 AT %QX1.4: BOOL;
	Y15 AT %QX1.5: BOOL;
	// 启动按钮LED
	Y16 AT %QX1.6: BOOL;
	// 停止按钮LED
	Y17 AT %QX1.7: BOOL;
	// 复位按钮LED
	Y20 AT %QX2.0: BOOL;
	Y21 AT %QX2.1: BOOL;
	// 下料传送带
	Y22 AT %QX2.2: BOOL;
	// 三色灯红
	Y23 AT %QX2.3: BOOL;
	// 三色灯黄
	Y24 AT %QX2.4: BOOL;
	// 三色灯绿
	Y25 AT %QX2.5: BOOL;
	// 三色灯蜂鸣
	Y26 AT %QX2.6: BOOL;
	// 联机卡盘夹紧
	Y27 AT %QX2.7: BOOL;
	// 联机启动
	Y30 AT %QX3.0: BOOL;
	// 联机停止
	Y31 AT %QX3.1: BOOL;
	Y32 AT %QX3.2: BOOL;
	Y33 AT %QX3.3: BOOL;
	Y34 AT %QX3.4: BOOL;
	Y35 AT %QX3.5: BOOL;
	Y36 AT %QX3.6: BOOL;
	Y37 AT %QX3.7: BOOL;
END_VAR

// Device/Application/PLC_PRG
PROGRAM PLC_PRG

END_PROGRAM

// Device/Application/FunctionBlock/Public_Prog
PROGRAM Public_Prog
VAR
	Clock_10Hz: FB102_ClockPuls;
	Clock_5Hz: FB102_ClockPuls;
	Clock_2Hz: FB102_ClockPuls;
	Clock_1Hz: FB102_ClockPuls;
	Clock_HalfHz: FB102_ClockPuls;
END_VAR
VAR // added by the converter: edge detectors and wires of the graphical bodies
    _rt1 : R_TRIG;
END_VAR

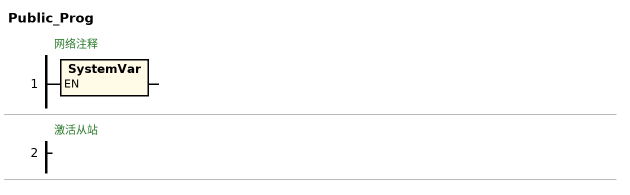
// NETWORK 1
// 网络注释
SystemVar();

// NETWORK 2
// 激活从站

ACTION SystemVar:
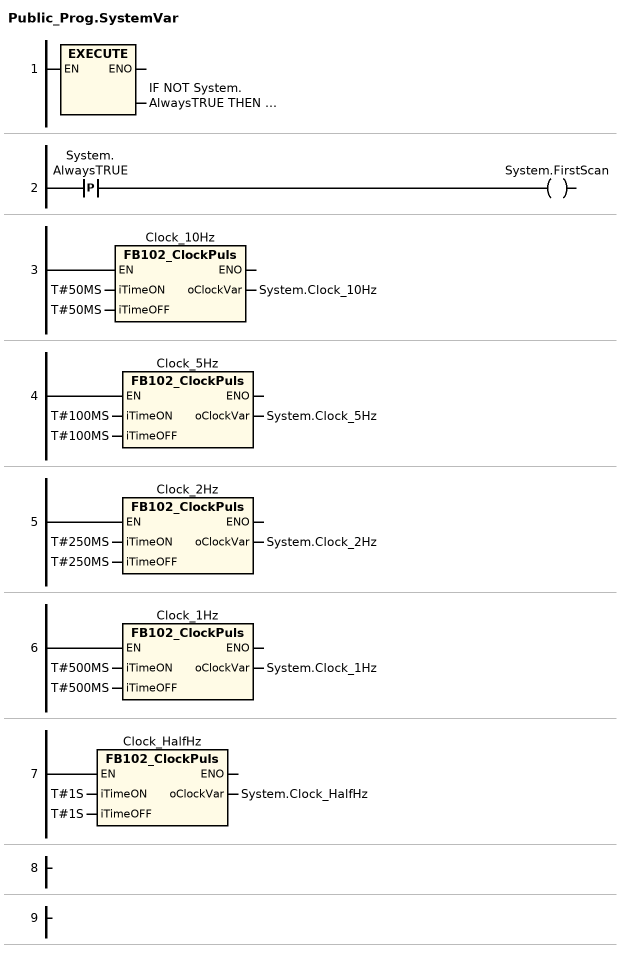
// NETWORK 1
IF NOT System.AlwaysTRUE THEN
	System.AlwaysTRUE := TRUE;
END_IF
IF  System.AlwaysFALSE THEN
	System.AlwaysFALSE := FALSE;
END_IF
IF NOT Publics.CYGIA_ON THEN
	Publics.CYGIA_ON := TRUE;
END_IF
IF  Publics.CYGIA_OFF THEN
	Publics.CYGIA_OFF := FALSE;
END_IF

// NETWORK 2
_rt1(CLK := System.AlwaysTRUE);
System.FirstScan := _rt1.Q;

// NETWORK 3
Clock_10Hz(iTimeON := T#50MS, iTimeOFF := T#50MS, oClockVar => System.Clock_10Hz); // FB102_ClockPuls

// NETWORK 4
Clock_5Hz(iTimeON := T#100MS, iTimeOFF := T#100MS, oClockVar => System.Clock_5Hz); // FB102_ClockPuls

// NETWORK 5
Clock_2Hz(iTimeON := T#250MS, iTimeOFF := T#250MS, oClockVar => System.Clock_2Hz); // FB102_ClockPuls

// NETWORK 6
Clock_1Hz(iTimeON := T#500MS, iTimeOFF := T#500MS, oClockVar => System.Clock_1Hz); // FB102_ClockPuls

// NETWORK 7
Clock_HalfHz(iTimeON := T#1S, iTimeOFF := T#1S, oClockVar => System.Clock_HalfHz); // FB102_ClockPuls

// NETWORK 8

// NETWORK 9
END_ACTION

END_PROGRAM

// Device/Application/FunctionBlock/FB102_ClockPuls
FUNCTION_BLOCK FB102_ClockPuls
VAR_INPUT
	///脉冲ON时间
	iTimeON: TIME;
	///脉冲OFF时间
	iTimeOFF: TIME;
END_VAR
VAR_OUTPUT
	///时钟脉冲差速器
	oClockVar: BOOL;
END_VAR
VAR
	TON_Clock: TON;
	TOF_Clock: TOF;
END_VAR

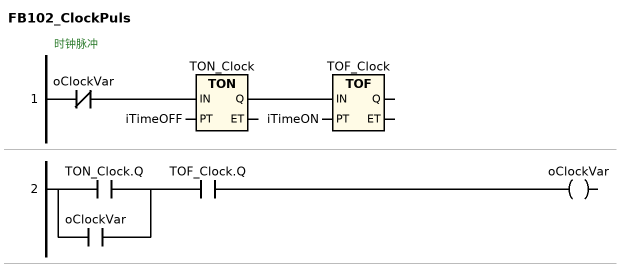
// NETWORK 1
// 时钟脉冲
TON_Clock(IN := NOT oClockVar, PT := iTimeOFF); // TON
TOF_Clock(IN := TON_Clock.Q, PT := iTimeON); // TOF

// NETWORK 2
oClockVar := (TON_Clock.Q OR oClockVar) AND TOF_Clock.Q;

END_FUNCTION_BLOCK

// Device/Application/信号
PROGRAM 信号
VAR
	循环时间传递: BOOL;
	循环时间: WORD;
	P2_Y下极限: REAL;
	P2_Y上极限: REAL;
	P2_X下极限: REAL;
	P2_X上极限: REAL;
	允许自动运行: BOOL;
	P2_Z1上极限: REAL;
	P2_Z1下极限: REAL;
	P2_Z2上极限: REAL;
	P2_Z2下极限: REAL;
	P2范围内: BOOL;
	TON_0: TON;
	循环停止通知: BOOL;
	P1: 点位范围判断;
	点位范围判断_0: 点位范围判断;
	点位范围判断_1: 点位范围判断;
	点位范围判断_2: 点位范围判断;
	点位范围判断_3: 点位范围判断;
	点位范围判断_4: 点位范围判断;
	点位范围判断_5: 点位范围判断;
	点位范围判断_6: 点位范围判断;
	点位范围判断_7: 点位范围判断;
	BLINK_0: BLINK;
	上次循环时间: WORD;
END_VAR
VAR // added by the converter: edge detectors and wires of the graphical bodies
    _w1 : BOOL;
    _rt1, _rt2 : R_TRIG;
END_VAR

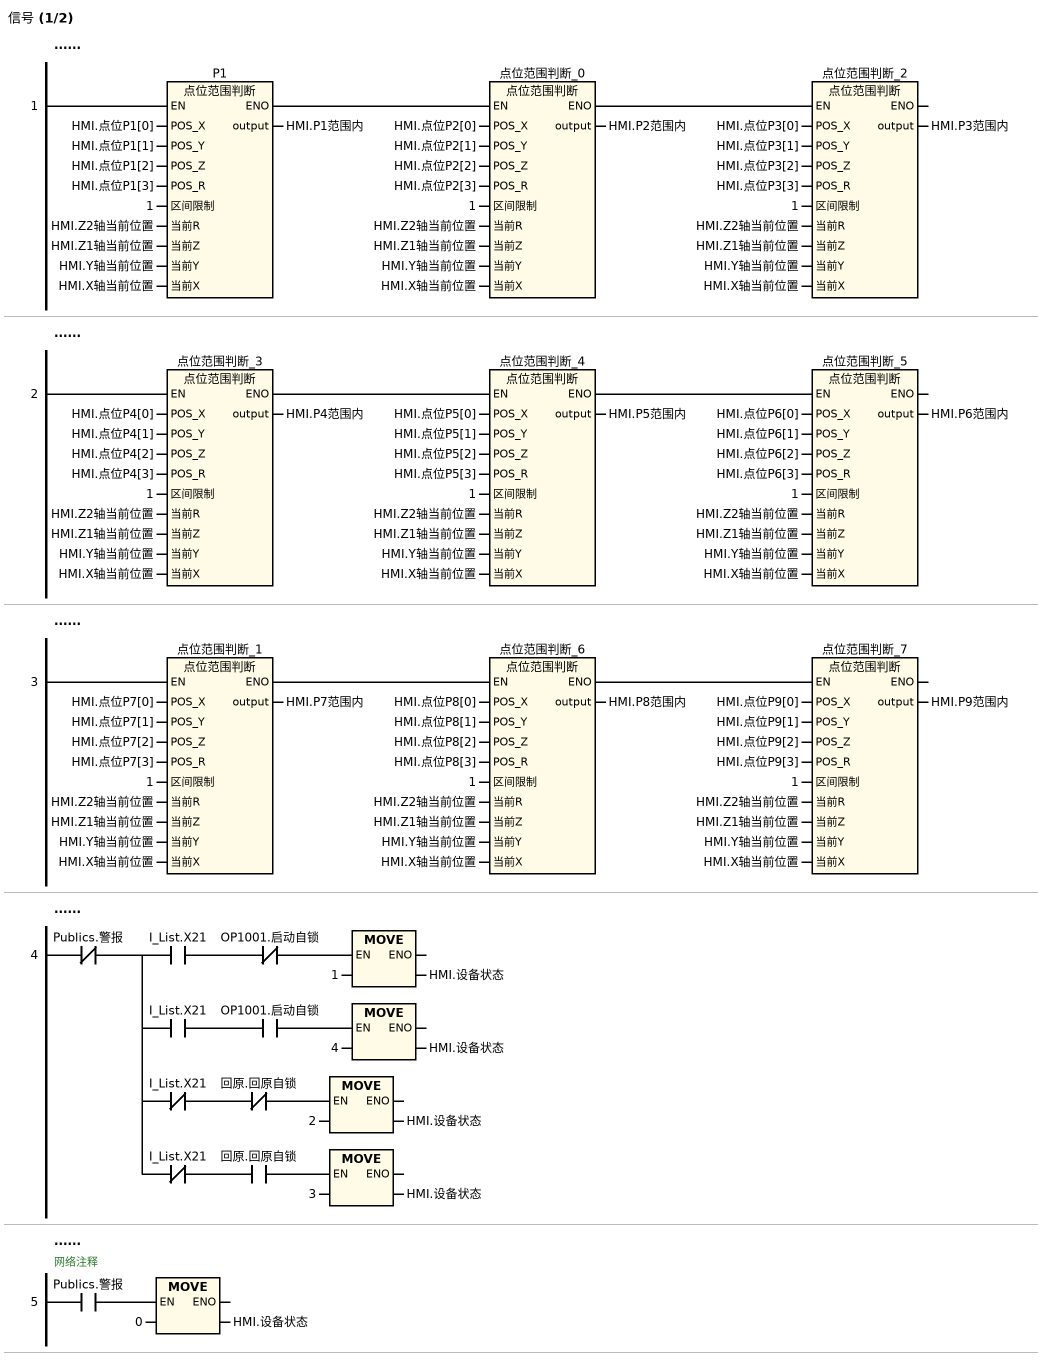
// NETWORK 1: ......
P1(
    POS_X := HMI.点位P1[0],
    POS_Y := HMI.点位P1[1],
    POS_Z := HMI.点位P1[2],
    POS_R := HMI.点位P1[3],
    区间限制 := 1,
    当前R := HMI.Z2轴当前位置,
    当前Z := HMI.Z1轴当前位置,
    当前Y := HMI.Y轴当前位置,
    当前X := HMI.X轴当前位置,
    output => HMI.P1范围内); // 点位范围判断
点位范围判断_0(
    POS_X := HMI.点位P2[0],
    POS_Y := HMI.点位P2[1],
    POS_Z := HMI.点位P2[2],
    POS_R := HMI.点位P2[3],
    区间限制 := 1,
    当前R := HMI.Z2轴当前位置,
    当前Z := HMI.Z1轴当前位置,
    当前Y := HMI.Y轴当前位置,
    当前X := HMI.X轴当前位置,
    output => HMI.P2范围内); // 点位范围判断
点位范围判断_2(
    POS_X := HMI.点位P3[0],
    POS_Y := HMI.点位P3[1],
    POS_Z := HMI.点位P3[2],
    POS_R := HMI.点位P3[3],
    区间限制 := 1,
    当前R := HMI.Z2轴当前位置,
    当前Z := HMI.Z1轴当前位置,
    当前Y := HMI.Y轴当前位置,
    当前X := HMI.X轴当前位置,
    output => HMI.P3范围内); // 点位范围判断

// NETWORK 2: ......
点位范围判断_3(
    POS_X := HMI.点位P4[0],
    POS_Y := HMI.点位P4[1],
    POS_Z := HMI.点位P4[2],
    POS_R := HMI.点位P4[3],
    区间限制 := 1,
    当前R := HMI.Z2轴当前位置,
    当前Z := HMI.Z1轴当前位置,
    当前Y := HMI.Y轴当前位置,
    当前X := HMI.X轴当前位置,
    output => HMI.P4范围内); // 点位范围判断
点位范围判断_4(
    POS_X := HMI.点位P5[0],
    POS_Y := HMI.点位P5[1],
    POS_Z := HMI.点位P5[2],
    POS_R := HMI.点位P5[3],
    区间限制 := 1,
    当前R := HMI.Z2轴当前位置,
    当前Z := HMI.Z1轴当前位置,
    当前Y := HMI.Y轴当前位置,
    当前X := HMI.X轴当前位置,
    output => HMI.P5范围内); // 点位范围判断
点位范围判断_5(
    POS_X := HMI.点位P6[0],
    POS_Y := HMI.点位P6[1],
    POS_Z := HMI.点位P6[2],
    POS_R := HMI.点位P6[3],
    区间限制 := 1,
    当前R := HMI.Z2轴当前位置,
    当前Z := HMI.Z1轴当前位置,
    当前Y := HMI.Y轴当前位置,
    当前X := HMI.X轴当前位置,
    output => HMI.P6范围内); // 点位范围判断

// NETWORK 3: ......
点位范围判断_1(
    POS_X := HMI.点位P7[0],
    POS_Y := HMI.点位P7[1],
    POS_Z := HMI.点位P7[2],
    POS_R := HMI.点位P7[3],
    区间限制 := 1,
    当前R := HMI.Z2轴当前位置,
    当前Z := HMI.Z1轴当前位置,
    当前Y := HMI.Y轴当前位置,
    当前X := HMI.X轴当前位置,
    output => HMI.P7范围内); // 点位范围判断
点位范围判断_6(
    POS_X := HMI.点位P8[0],
    POS_Y := HMI.点位P8[1],
    POS_Z := HMI.点位P8[2],
    POS_R := HMI.点位P8[3],
    区间限制 := 1,
    当前R := HMI.Z2轴当前位置,
    当前Z := HMI.Z1轴当前位置,
    当前Y := HMI.Y轴当前位置,
    当前X := HMI.X轴当前位置,
    output => HMI.P8范围内); // 点位范围判断
点位范围判断_7(
    POS_X := HMI.点位P9[0],
    POS_Y := HMI.点位P9[1],
    POS_Z := HMI.点位P9[2],
    POS_R := HMI.点位P9[3],
    区间限制 := 1,
    当前R := HMI.Z2轴当前位置,
    当前Z := HMI.Z1轴当前位置,
    当前Y := HMI.Y轴当前位置,
    当前X := HMI.X轴当前位置,
    output => HMI.P9范围内); // 点位范围判断

// NETWORK 4: ......
_w1 := NOT Publics.警报;
IF _w1 AND I_List.X21 AND NOT OP1001.启动自锁 THEN HMI.设备状态 := 1; END_IF
IF _w1 AND I_List.X21 AND OP1001.启动自锁 THEN HMI.设备状态 := 4; END_IF
IF _w1 AND NOT I_List.X21 AND NOT 回原.回原自锁 THEN HMI.设备状态 := 2; END_IF
IF _w1 AND NOT I_List.X21 AND 回原.回原自锁 THEN HMI.设备状态 := 3; END_IF

// NETWORK 5: ......
// 网络注释
IF Publics.警报 THEN HMI.设备状态 := 0; END_IF

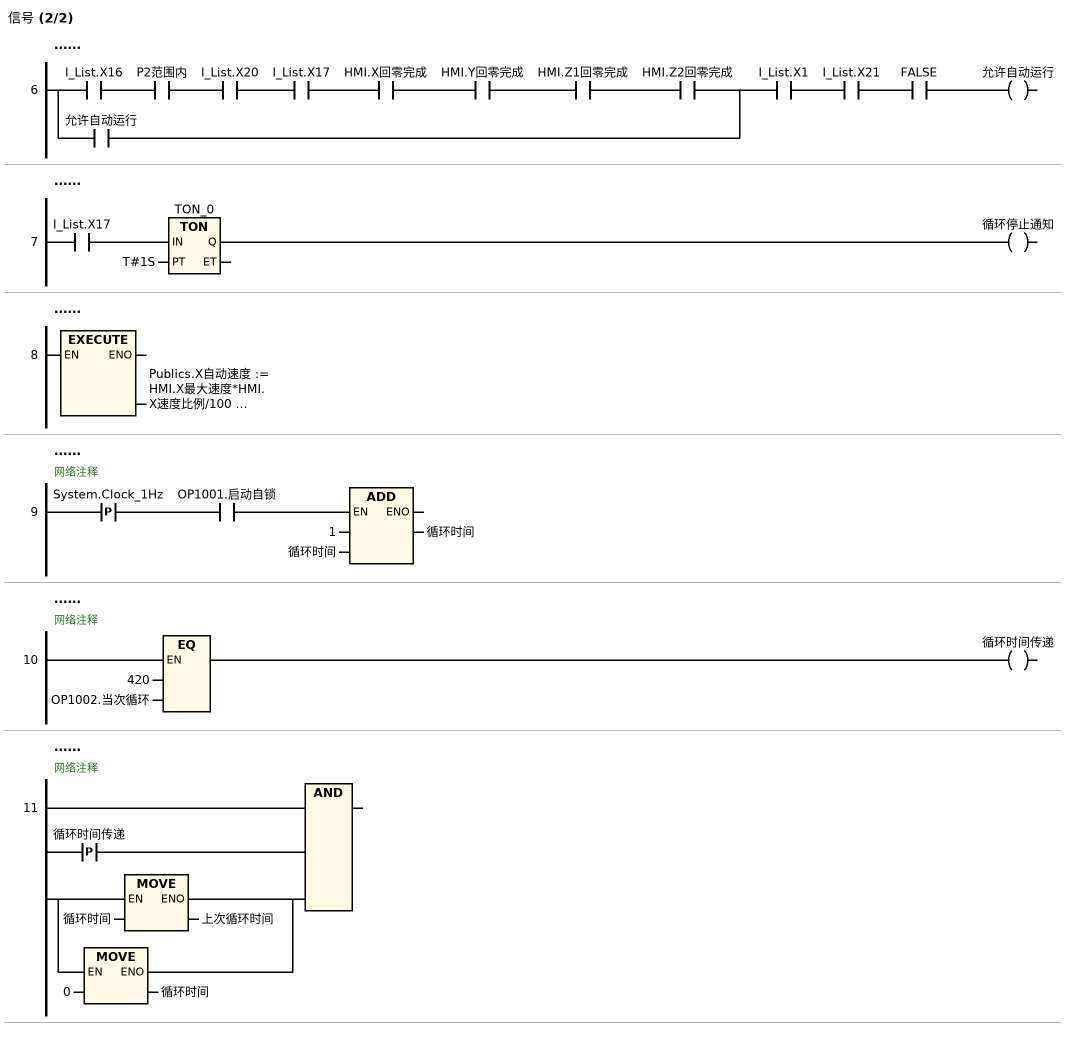
// NETWORK 6: ......
允许自动运行 := (I_List.X16 AND P2范围内 AND I_List.X20 AND I_List.X17 AND HMI.X回零完成 AND HMI.Y回零完成 AND HMI.Z1回零完成 AND HMI.Z2回零完成 OR 允许自动运行) AND I_List.X1 AND I_List.X21 AND FALSE;

// NETWORK 7: ......
TON_0(IN := I_List.X17, PT := T#1S); // TON
循环停止通知 := TON_0.Q;

// NETWORK 8: ......
Publics.X自动速度 := HMI.X最大速度*HMI.X速度比例/100;
Publics.Y自动速度 := HMI.Y最大速度*HMI.Y速度比例/100;
Publics.Z1自动速度 := HMI.Z1最大速度*HMI.Z1速度比例/100;
Publics.Z2自动速度 := HMI.Z2最大速度*HMI.Z2速度比例/100;

// NETWORK 9: ......
// 网络注释
_rt1(CLK := System.Clock_1Hz);
IF _rt1.Q AND OP1001.启动自锁 THEN 循环时间 := 1 + 循环时间; END_IF

// NETWORK 10: ......
// 网络注释
循环时间传递 := 420 = OP1002.当次循环;

// NETWORK 11: ......
// 网络注释
_rt2(CLK := 循环时间传递);
上次循环时间 := 循环时间;
循环时间 := 0;
(* _rt2.Q AND (TRUE OR TRUE); result not used *)

END_PROGRAM

// Device/Application/FunctionBlock/点位范围判断
FUNCTION_BLOCK 点位范围判断
VAR_INPUT
	POS_X: REAL;
	POS_Y: REAL;
	POS_Z: REAL;
	POS_R: REAL;
END_VAR
VAR
	X上极限: REAL;
	X下极限: REAL;
	Y上极限: REAL;
	Y下极限: REAL;
	R上极限: REAL;
	R下极限: REAL;
	Z上极限: REAL;
	Z下极限: REAL;
END_VAR
VAR_OUTPUT
	output: BOOL;
END_VAR
VAR_INPUT
	区间限制: REAL;
	当前R: REAL;
	当前Z: REAL;
	当前Y: REAL;
	当前X: REAL;
END_VAR

X上极限:=POS_X+区间限制;
X下极限:=POS_X-区间限制;
Y上极限:=POS_Y+区间限制;
Y下极限:=POS_Y-区间限制;
R上极限:=POS_Z+区间限制;
R下极限:=POS_Z-区间限制;
Z上极限:=POS_R+区间限制;
Z下极限:=POS_R-区间限制;
IF X上极限>当前X THEN
    IF X下极限<当前X THEN
		IF Y上极限>当前Y THEN
			IF Y下极限<当前Y THEN
				IF R上极限>当前R THEN
					IF R下极限<当前R THEN
						IF Z上极限>当前Z THEN
							IF Z下极限<当前Z THEN
								output:=1;	
							ELSE
								output:=0;		
							END_IF
						ELSE
							output:=0;	
						END_IF
					ELSE
						output:=0;	
					END_IF
				ELSE
					output:=0;
				END_IF
			ELSE
				output:=0;
			END_IF
		ELSE
			output:=0;
		END_IF
	ELSE
		output:=0;
	END_IF
ELSE
	output:=0;
END_IF

END_FUNCTION_BLOCK

// Device/Application/OP1001
PROGRAM OP1001
VAR
	启动自锁: BOOL;
	下次循环: word;
	当次循环: word;
	循环停止: BOOL;
	阻止运行条件: BOOL;
	TON_0: TON;
	TON_1: TON;
	TON_2: TON;
	通知_允许抓取物料: BOOL;
	A1: BOOL;
	A2: BOOL;
	A3: BOOL;
	A4: BOOL;
	A5: BOOL;
	A6: BOOL;
	A7: BOOL;
	A8: BOOL;
	启动条件: BOOL;
	DEBUG: BOOL;
END_VAR
VAR_INPUT
	通知_物料抓取完成: BOOL;
END_VAR
VAR
	流程结束: BOOL;
END_VAR
VAR // added by the converter: edge detectors and wires of the graphical bodies
    _w1, _w2, _w3, _w4, _w5, _w6, _w7, _w8 : BOOL;
    _rt1, _rt2 : R_TRIG;
END_VAR

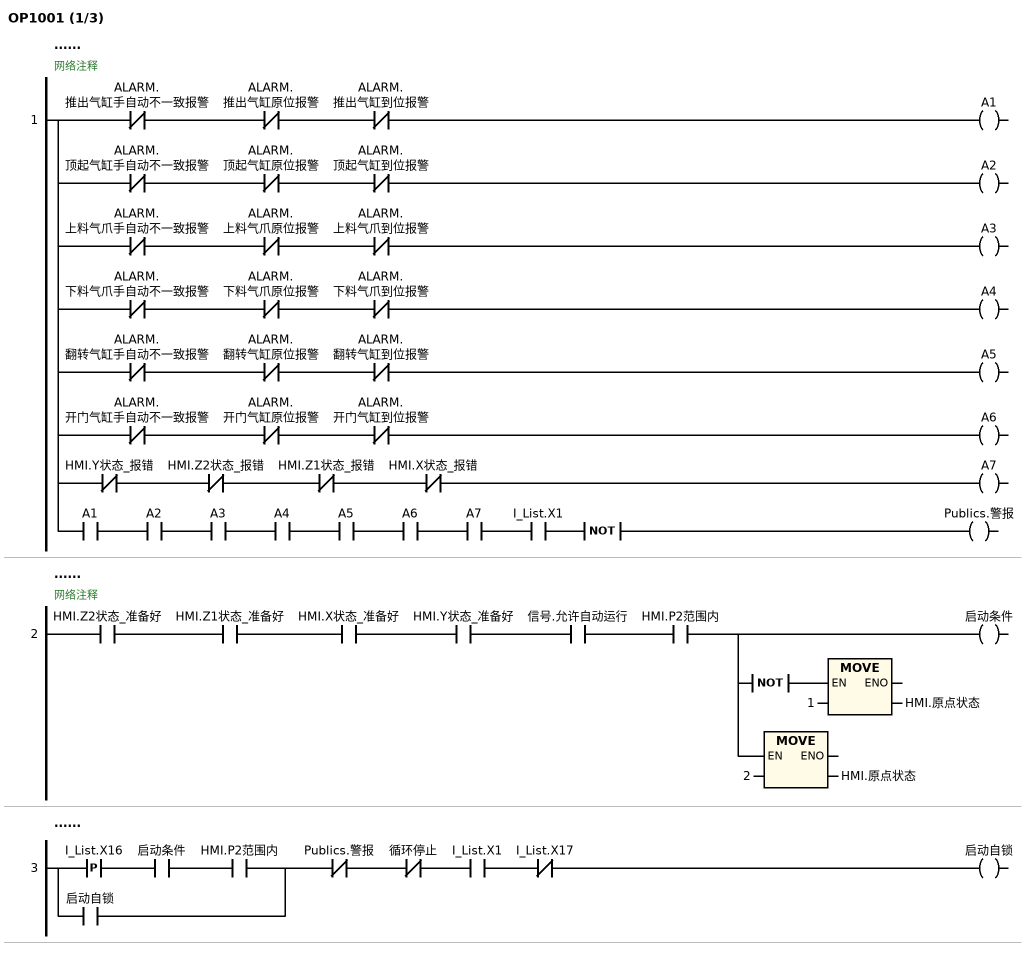
// NETWORK 1: ......
// 网络注释
A1 := NOT ALARM.推出气缸手自动不一致报警 AND NOT ALARM.推出气缸原位报警 AND NOT ALARM.推出气缸到位报警;
A2 := NOT ALARM.顶起气缸手自动不一致报警 AND NOT ALARM.顶起气缸原位报警 AND NOT ALARM.顶起气缸到位报警;
A3 := NOT ALARM.上料气爪手自动不一致报警 AND NOT ALARM.上料气爪原位报警 AND NOT ALARM.上料气爪到位报警;
A4 := NOT ALARM.下料气爪手自动不一致报警 AND NOT ALARM.下料气爪原位报警 AND NOT ALARM.下料气爪到位报警;
A5 := NOT ALARM.翻转气缸手自动不一致报警 AND NOT ALARM.翻转气缸原位报警 AND NOT ALARM.翻转气缸到位报警;
A6 := NOT ALARM.开门气缸手自动不一致报警 AND NOT ALARM.开门气缸原位报警 AND NOT ALARM.开门气缸到位报警;
A7 := NOT HMI.Y状态_报错 AND NOT HMI.Z2状态_报错 AND NOT HMI.Z1状态_报错 AND NOT HMI.X状态_报错;
Publics.警报 := NOT (A1 AND A2 AND A3 AND A4 AND A5 AND A6 AND A7 AND I_List.X1);

// NETWORK 2: ......
// 网络注释
_w1 := HMI.Z2状态_准备好 AND HMI.Z1状态_准备好 AND HMI.X状态_准备好 AND HMI.Y状态_准备好 AND 信号.允许自动运行 AND HMI.P2范围内;
启动条件 := _w1;
IF NOT _w1 THEN HMI.原点状态 := 1; END_IF
IF _w1 THEN HMI.原点状态 := 2; END_IF

// NETWORK 3: ......
_rt1(CLK := I_List.X16);
启动自锁 := (_rt1.Q AND 启动条件 AND HMI.P2范围内 OR 启动自锁) AND NOT Publics.警报 AND NOT 循环停止 AND I_List.X1 AND NOT I_List.X17;

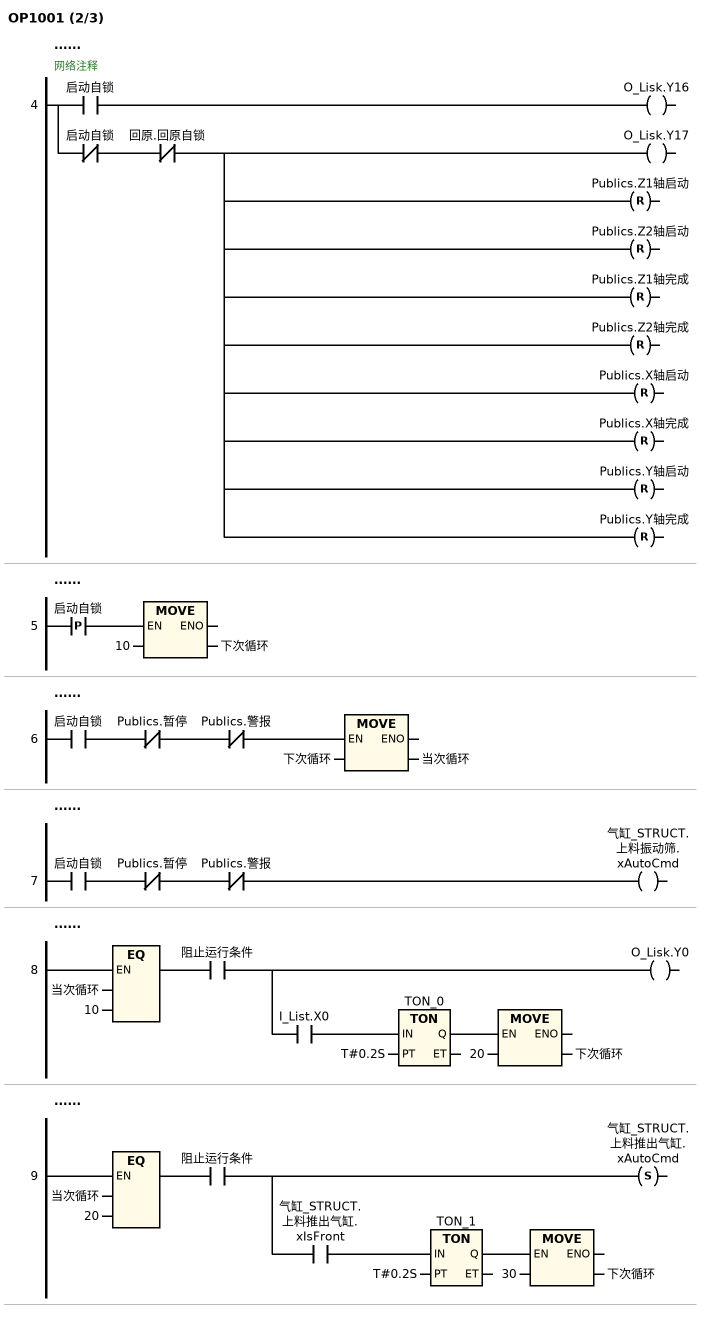
// NETWORK 4: ......
// 网络注释
O_Lisk.Y16 := 启动自锁;
_w2 := NOT 启动自锁 AND NOT 回原.回原自锁;
O_Lisk.Y17 := _w2;
Publics.Z1轴启动 R= _w2;
Publics.Z2轴启动 R= _w2;
Publics.Z1轴完成 R= _w2;
Publics.Z2轴完成 R= _w2;
Publics.X轴启动 R= _w2;
Publics.X轴完成 R= _w2;
Publics.Y轴启动 R= _w2;
Publics.Y轴完成 R= _w2;

// NETWORK 5: ......
_rt2(CLK := 启动自锁);
IF _rt2.Q THEN 下次循环 := 10; END_IF

// NETWORK 6: ......
IF 启动自锁 AND NOT Publics.暂停 AND NOT Publics.警报 THEN 当次循环 := 下次循环; END_IF

// NETWORK 7: ......
气缸_STRUCT.上料振动筛.xAutoCmd := 启动自锁 AND NOT Publics.暂停 AND NOT Publics.警报;

// NETWORK 8: ......
_w3 := 当次循环 = 10 AND 阻止运行条件;
O_Lisk.Y0 := _w3;
TON_0(IN := _w3 AND I_List.X0, PT := T#0.2S); // TON
IF TON_0.Q THEN 下次循环 := 20; END_IF

// NETWORK 9: ......
_w4 := 当次循环 = 20 AND 阻止运行条件;
气缸_STRUCT.上料推出气缸.xAutoCmd S= _w4;
TON_1(IN := _w4 AND 气缸_STRUCT.上料推出气缸.xIsFront, PT := T#0.2S); // TON
IF TON_1.Q THEN 下次循环 := 30; END_IF

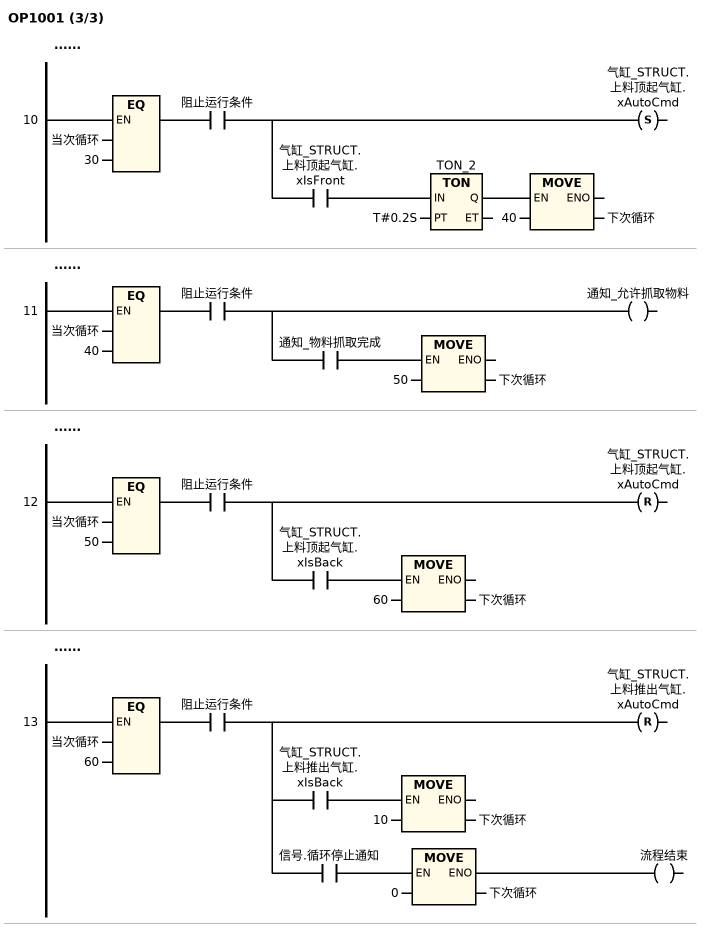
// NETWORK 10: ......
_w5 := 当次循环 = 30 AND 阻止运行条件;
气缸_STRUCT.上料顶起气缸.xAutoCmd S= _w5;
TON_2(IN := _w5 AND 气缸_STRUCT.上料顶起气缸.xIsFront, PT := T#0.2S); // TON
IF TON_2.Q THEN 下次循环 := 40; END_IF

// NETWORK 11: ......
_w6 := 当次循环 = 40 AND 阻止运行条件;
通知_允许抓取物料 := _w6;
IF _w6 AND 通知_物料抓取完成 THEN 下次循环 := 50; END_IF

// NETWORK 12: ......
_w7 := 当次循环 = 50 AND 阻止运行条件;
气缸_STRUCT.上料顶起气缸.xAutoCmd R= _w7;
IF _w7 AND 气缸_STRUCT.上料顶起气缸.xIsBack THEN 下次循环 := 60; END_IF

// NETWORK 13: ......
_w8 := 当次循环 = 60 AND 阻止运行条件;
气缸_STRUCT.上料推出气缸.xAutoCmd R= _w8;
IF _w8 AND 气缸_STRUCT.上料推出气缸.xIsBack THEN 下次循环 := 10; END_IF
IF _w8 AND 信号.循环停止通知 THEN 下次循环 := 0; END_IF
流程结束 := _w8 AND 信号.循环停止通知;

END_PROGRAM

// Device/Application/回原
PROGRAM 回原
VAR
	下次循环: WORD;
	回原条件: BOOL;
	阻止条件: BOOL;
	回原自锁: BOOL;
	当次循环: WORD;
	判断下极限: REAL;
	判断上极限: REAL;
	避开扫描周期: BOOL;
	流程结束: BOOL;
END_VAR
VAR // added by the converter: edge detectors and wires of the graphical bodies
    _rt1 : R_TRIG;
    _w1, _w2, _w3, _w4, _w5, _w6, _w7, _w8, _w9, _w10, _w11, _w12 : BOOL;
END_VAR

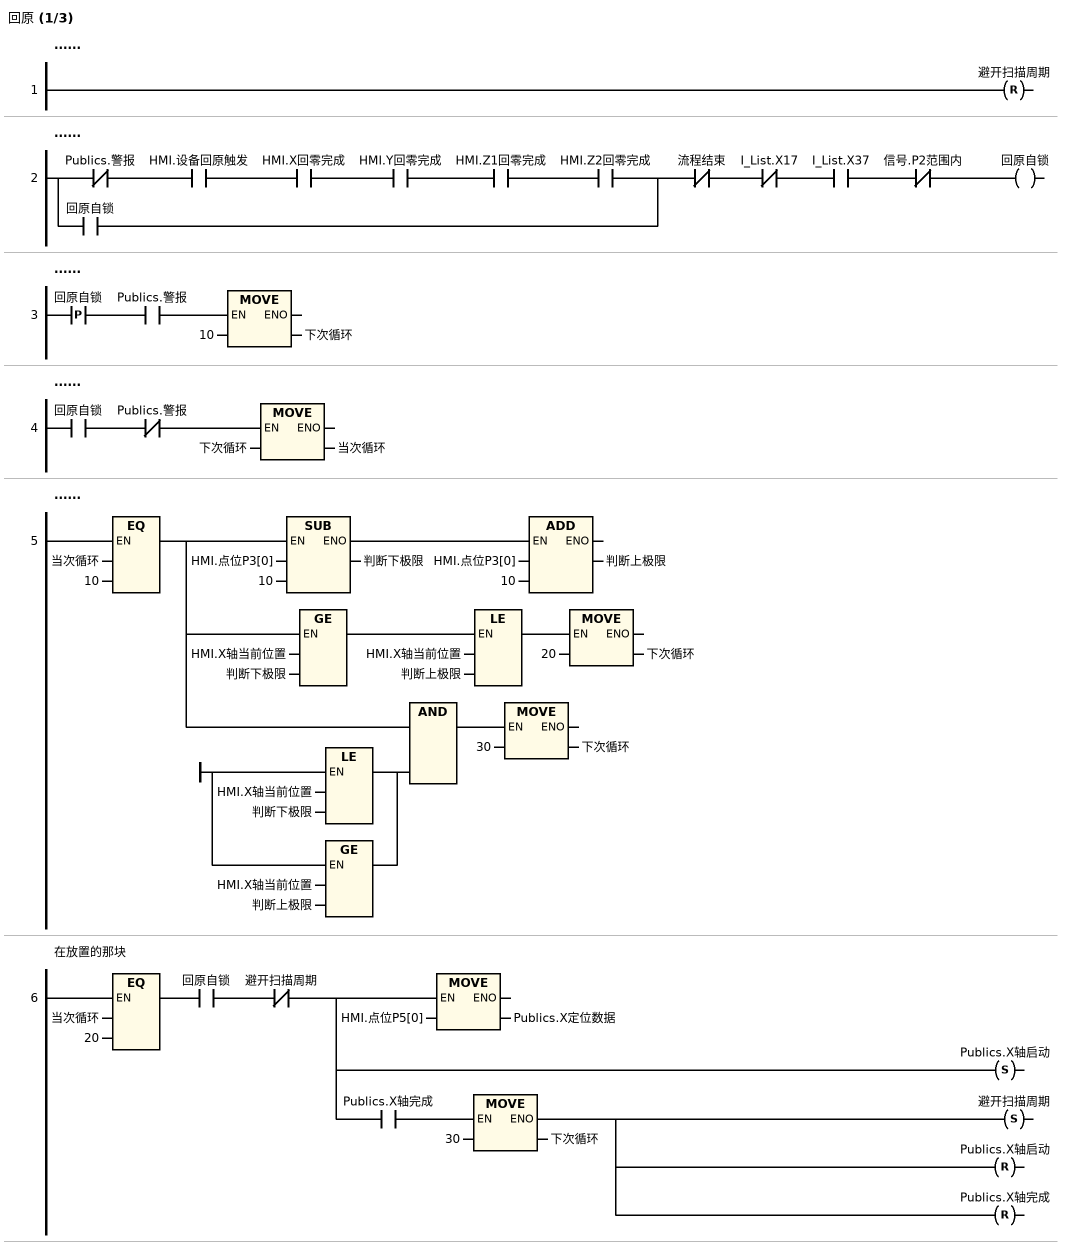
// NETWORK 1: ......
避开扫描周期 R= TRUE;

// NETWORK 2: ......
回原自锁 := (NOT Publics.警报 AND HMI.设备回原触发 AND HMI.X回零完成 AND HMI.Y回零完成 AND HMI.Z1回零完成 AND HMI.Z2回零完成 OR 回原自锁) AND NOT 流程结束 AND NOT I_List.X17 AND I_List.X37 AND NOT 信号.P2范围内;

// NETWORK 3: ......
_rt1(CLK := 回原自锁);
IF _rt1.Q AND Publics.警报 THEN 下次循环 := 10; END_IF

// NETWORK 4: ......
IF 回原自锁 AND NOT Publics.警报 THEN 当次循环 := 下次循环; END_IF

// NETWORK 5: ......
_w1 := 当次循环 = 10;
IF _w1 THEN 判断下极限 := HMI.点位P3[0] - 10; END_IF
IF _w1 THEN 判断上极限 := HMI.点位P3[0] + 10; END_IF
IF _w1 AND HMI.X轴当前位置 >= 判断下极限 AND HMI.X轴当前位置 <= 判断上极限 THEN 下次循环 := 20; END_IF
IF _w1 AND (HMI.X轴当前位置 <= 判断下极限 OR HMI.X轴当前位置 >= 判断上极限) THEN 下次循环 := 30; END_IF

// NETWORK 6: 在放置的那块
_w2 := 当次循环 = 20 AND 回原自锁 AND NOT 避开扫描周期;
IF _w2 THEN Publics.X定位数据 := HMI.点位P5[0]; END_IF
Publics.X轴启动 S= _w2;
IF _w2 AND Publics.X轴完成 THEN 下次循环 := 30; END_IF
_w3 := _w2 AND Publics.X轴完成;
避开扫描周期 S= _w3;
Publics.X轴启动 R= _w3;
Publics.X轴完成 R= _w3;

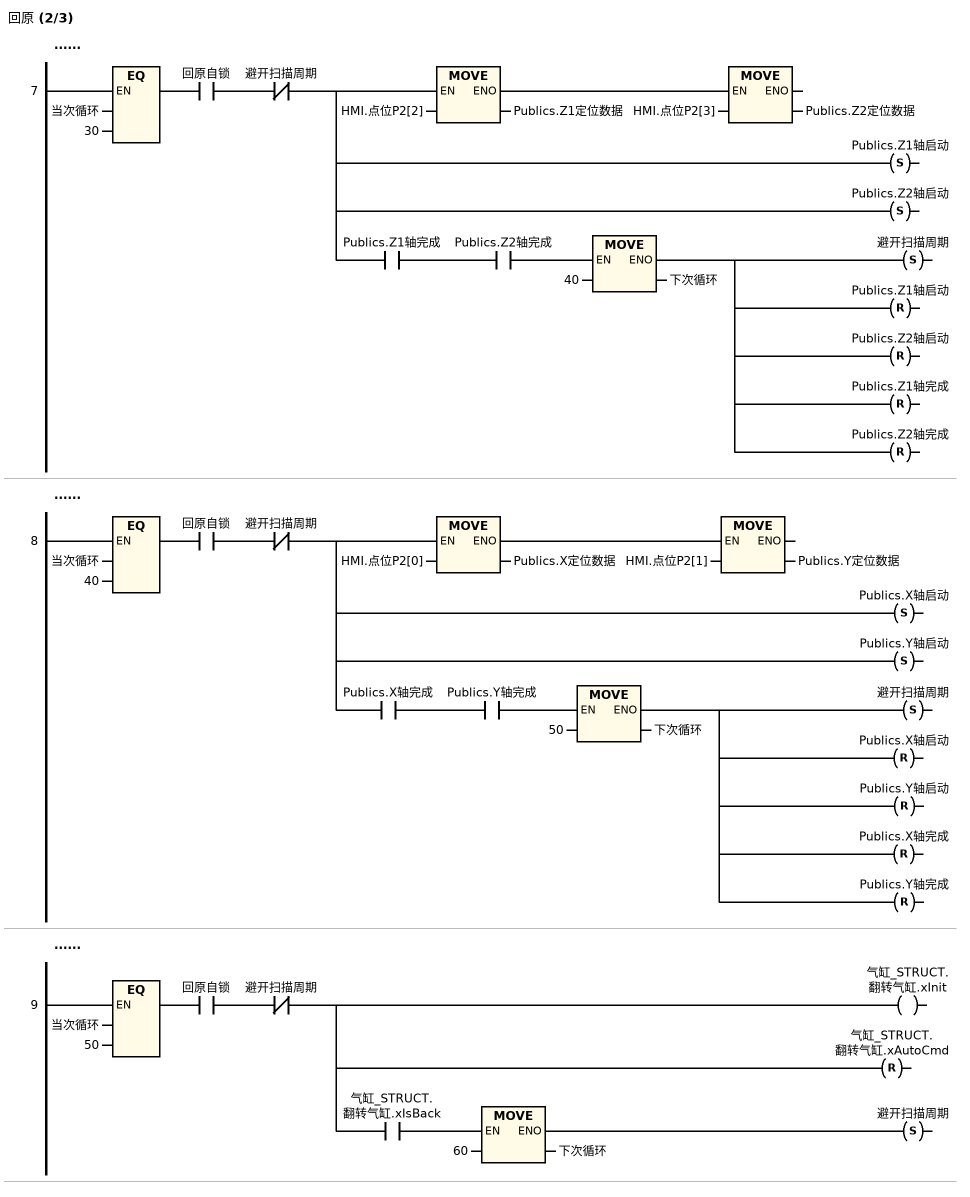
// NETWORK 7: ......
_w4 := 当次循环 = 30 AND 回原自锁 AND NOT 避开扫描周期;
IF _w4 THEN Publics.Z1定位数据 := HMI.点位P2[2]; END_IF
IF _w4 THEN Publics.Z2定位数据 := HMI.点位P2[3]; END_IF
Publics.Z1轴启动 S= _w4;
Publics.Z2轴启动 S= _w4;
IF _w4 AND Publics.Z1轴完成 AND Publics.Z2轴完成 THEN 下次循环 := 40; END_IF
_w5 := _w4 AND Publics.Z1轴完成 AND Publics.Z2轴完成;
避开扫描周期 S= _w5;
Publics.Z1轴启动 R= _w5;
Publics.Z2轴启动 R= _w5;
Publics.Z1轴完成 R= _w5;
Publics.Z2轴完成 R= _w5;

// NETWORK 8: ......
_w6 := 当次循环 = 40 AND 回原自锁 AND NOT 避开扫描周期;
IF _w6 THEN Publics.X定位数据 := HMI.点位P2[0]; END_IF
IF _w6 THEN Publics.Y定位数据 := HMI.点位P2[1]; END_IF
Publics.X轴启动 S= _w6;
Publics.Y轴启动 S= _w6;
IF _w6 AND Publics.X轴完成 AND Publics.Y轴完成 THEN 下次循环 := 50; END_IF
_w7 := _w6 AND Publics.X轴完成 AND Publics.Y轴完成;
避开扫描周期 S= _w7;
Publics.X轴启动 R= _w7;
Publics.Y轴启动 R= _w7;
Publics.X轴完成 R= _w7;
Publics.Y轴完成 R= _w7;

// NETWORK 9: ......
_w8 := 当次循环 = 50 AND 回原自锁 AND NOT 避开扫描周期;
气缸_STRUCT.翻转气缸.xInit := _w8;
气缸_STRUCT.翻转气缸.xAutoCmd R= _w8;
IF _w8 AND 气缸_STRUCT.翻转气缸.xIsBack THEN 下次循环 := 60; END_IF
避开扫描周期 S= _w8 AND 气缸_STRUCT.翻转气缸.xIsBack;

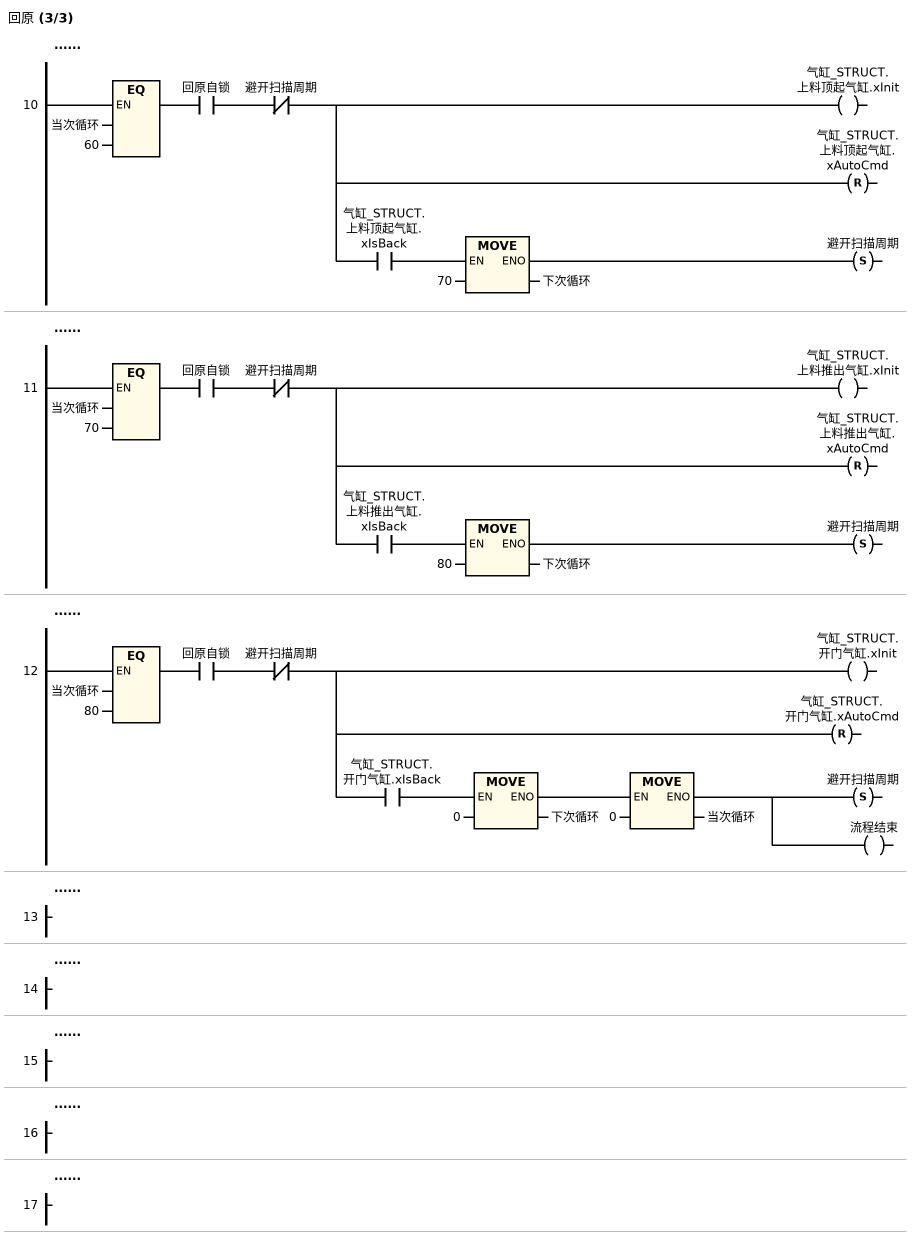
// NETWORK 10: ......
_w9 := 当次循环 = 60 AND 回原自锁 AND NOT 避开扫描周期;
气缸_STRUCT.上料顶起气缸.xInit := _w9;
气缸_STRUCT.上料顶起气缸.xAutoCmd R= _w9;
IF _w9 AND 气缸_STRUCT.上料顶起气缸.xIsBack THEN 下次循环 := 70; END_IF
避开扫描周期 S= _w9 AND 气缸_STRUCT.上料顶起气缸.xIsBack;

// NETWORK 11: ......
_w10 := 当次循环 = 70 AND 回原自锁 AND NOT 避开扫描周期;
气缸_STRUCT.上料推出气缸.xInit := _w10;
气缸_STRUCT.上料推出气缸.xAutoCmd R= _w10;
IF _w10 AND 气缸_STRUCT.上料推出气缸.xIsBack THEN 下次循环 := 80; END_IF
避开扫描周期 S= _w10 AND 气缸_STRUCT.上料推出气缸.xIsBack;

// NETWORK 12: ......
_w11 := 当次循环 = 80 AND 回原自锁 AND NOT 避开扫描周期;
气缸_STRUCT.开门气缸.xInit := _w11;
气缸_STRUCT.开门气缸.xAutoCmd R= _w11;
IF _w11 AND 气缸_STRUCT.开门气缸.xIsBack THEN 下次循环 := 0; END_IF
IF _w11 AND 气缸_STRUCT.开门气缸.xIsBack THEN 当次循环 := 0; END_IF
_w12 := _w11 AND 气缸_STRUCT.开门气缸.xIsBack;
避开扫描周期 S= _w12;
流程结束 := _w12;

// NETWORK 13: ......

// NETWORK 14: ......

// NETWORK 15: ......

// NETWORK 16: ......

// NETWORK 17: ......

END_PROGRAM

// Device/Application/OP1002
PROGRAM OP1002
VAR
	启动自锁: BOOL;
	循环停止: BOOL;
	下次循环: word;
	当次循环: word;
	伺服停止0: BOOL;
	避开扫描周期: BOOL;
	阻止运行条件: BOOL;
	通知_抓手上方要开门: BOOL;
	通知_门打开完成: BOOL;
	通知_关门: BOOL;
	通知_门关上了: BOOL;
	Y30_联机自锁: BOOL;
	TON_0: TON;
	DEBUG: BOOL;
END_VAR
VAR // added by the converter: edge detectors and wires of the graphical bodies
    _rt1, _rt2, _rt3 : R_TRIG;
    _w1, _w2, _w3, _w4, _w5, _w6, _w7, _w8, _w9, _w10, _w11, _w12, _w13, _w14, _w15, _w16, _w17, _w18, _w19, _w20, _w21, _w22, _w23, _w24, _w25, _w26, _w27, _w28, _w29, _w30, _w31, _w32, _w33, _w34, _w35, _w36, _w37, _w38, _w39, _w40, _w41, _w42, _w43, _w44, _w45, _w46, _w47, _w48, _w49, _w50, _w51, _w52, _w53, _w54, _w55, _w56, _w57, _w58, _w59, _w60, _w61, _w62, _w63, _w64, _w65, _w66, _w67, _w68, _w69, _w70, _w71, _w72, _w73, _w74, _w75 : BOOL;
END_VAR

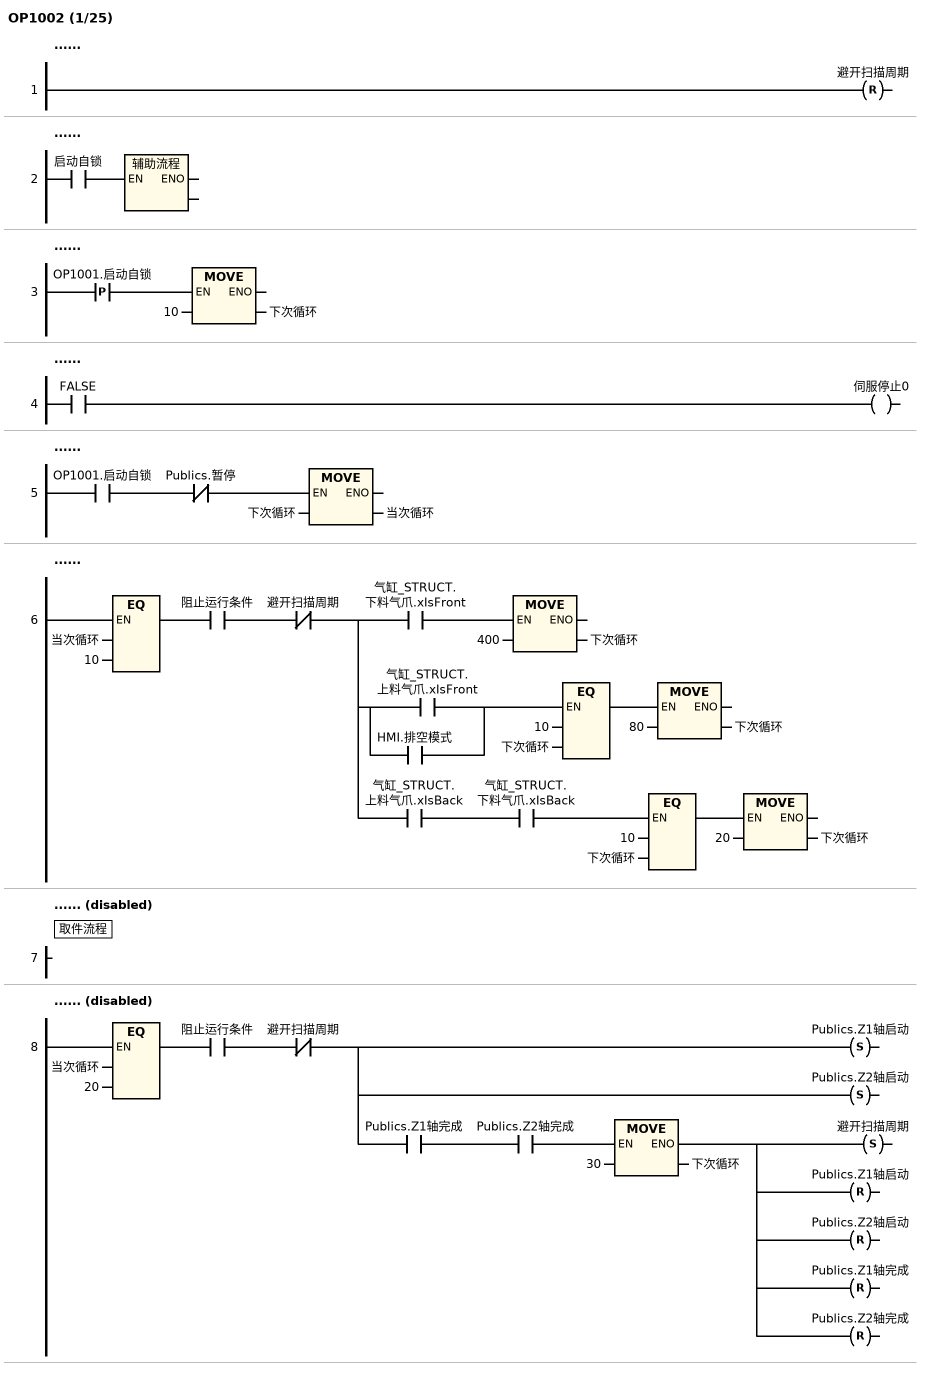
// NETWORK 1: ......
避开扫描周期 R= TRUE;

// NETWORK 2: ......
IF 启动自锁 THEN 辅助流程(); END_IF

// NETWORK 3: ......
_rt1(CLK := OP1001.启动自锁);
IF _rt1.Q THEN 下次循环 := 10; END_IF

// NETWORK 4: ......
伺服停止0 := FALSE;

// NETWORK 5: ......
IF OP1001.启动自锁 AND NOT Publics.暂停 THEN 当次循环 := 下次循环; END_IF

// NETWORK 6: ......
_w1 := 当次循环 = 10 AND 阻止运行条件 AND NOT 避开扫描周期;
IF _w1 AND 气缸_STRUCT.下料气爪.xIsFront THEN 下次循环 := 400; END_IF
IF _w1 AND (气缸_STRUCT.上料气爪.xIsFront OR HMI.排空模式) AND 10 = 下次循环 THEN 下次循环 := 80; END_IF
IF _w1 AND 气缸_STRUCT.上料气爪.xIsBack AND 气缸_STRUCT.下料气爪.xIsBack AND 10 = 下次循环 THEN 下次循环 := 20; END_IF

// NETWORK 7: ...... (disabled)
// label: 取件流程

// NETWORK 8: ...... (disabled)
// _w2 := 当次循环 = 20 AND 阻止运行条件 AND NOT 避开扫描周期;
// Publics.Z1轴启动 S= _w2;
// Publics.Z2轴启动 S= _w2;
// IF _w2 AND Publics.Z1轴完成 AND Publics.Z2轴完成 THEN 下次循环 := 30; END_IF
// _w3 := _w2 AND Publics.Z1轴完成 AND Publics.Z2轴完成;
// 避开扫描周期 S= _w3;
// Publics.Z1轴启动 R= _w3;
// Publics.Z2轴启动 R= _w3;
// Publics.Z1轴完成 R= _w3;
// Publics.Z2轴完成 R= _w3;

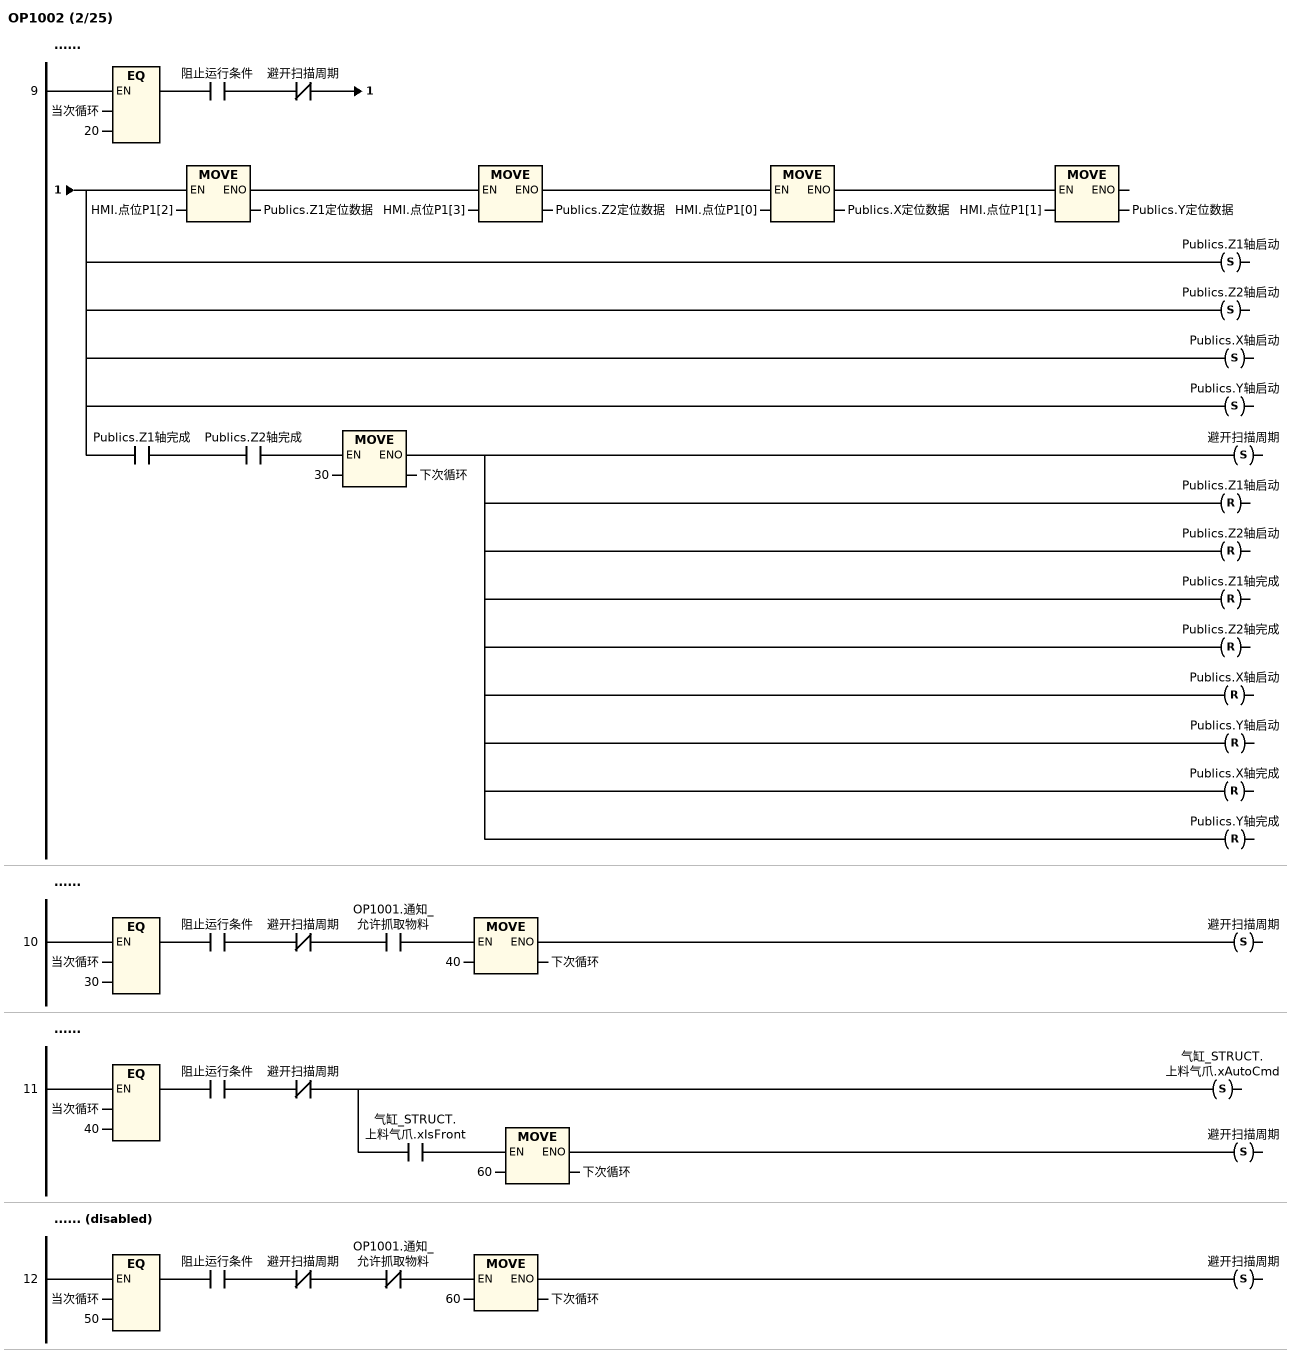
// NETWORK 9: ......
_w4 := 当次循环 = 20 AND 阻止运行条件 AND NOT 避开扫描周期;
IF _w4 THEN Publics.Z1定位数据 := HMI.点位P1[2]; END_IF
IF _w4 THEN Publics.Z2定位数据 := HMI.点位P1[3]; END_IF
IF _w4 THEN Publics.X定位数据 := HMI.点位P1[0]; END_IF
IF _w4 THEN Publics.Y定位数据 := HMI.点位P1[1]; END_IF
Publics.Z1轴启动 S= _w4;
Publics.Z2轴启动 S= _w4;
Publics.X轴启动 S= _w4;
Publics.Y轴启动 S= _w4;
IF _w4 AND Publics.Z1轴完成 AND Publics.Z2轴完成 THEN 下次循环 := 30; END_IF
_w5 := _w4 AND Publics.Z1轴完成 AND Publics.Z2轴完成;
避开扫描周期 S= _w5;
Publics.Z1轴启动 R= _w5;
Publics.Z2轴启动 R= _w5;
Publics.Z1轴完成 R= _w5;
Publics.Z2轴完成 R= _w5;
Publics.X轴启动 R= _w5;
Publics.Y轴启动 R= _w5;
Publics.X轴完成 R= _w5;
Publics.Y轴完成 R= _w5;

// NETWORK 10: ......
_w6 := 当次循环 = 30 AND 阻止运行条件 AND NOT 避开扫描周期 AND OP1001.通知_允许抓取物料;
IF _w6 THEN 下次循环 := 40; END_IF
避开扫描周期 S= _w6;

// NETWORK 11: ......
_w7 := 当次循环 = 40 AND 阻止运行条件 AND NOT 避开扫描周期;
气缸_STRUCT.上料气爪.xAutoCmd S= _w7;
IF _w7 AND 气缸_STRUCT.上料气爪.xIsFront THEN 下次循环 := 60; END_IF
避开扫描周期 S= _w7 AND 气缸_STRUCT.上料气爪.xIsFront;

// NETWORK 12: ...... (disabled)
// _w8 := 当次循环 = 50 AND 阻止运行条件 AND NOT 避开扫描周期 AND NOT OP1001.通知_允许抓取物料;
// IF _w8 THEN 下次循环 := 60; END_IF
// 避开扫描周期 S= _w8;

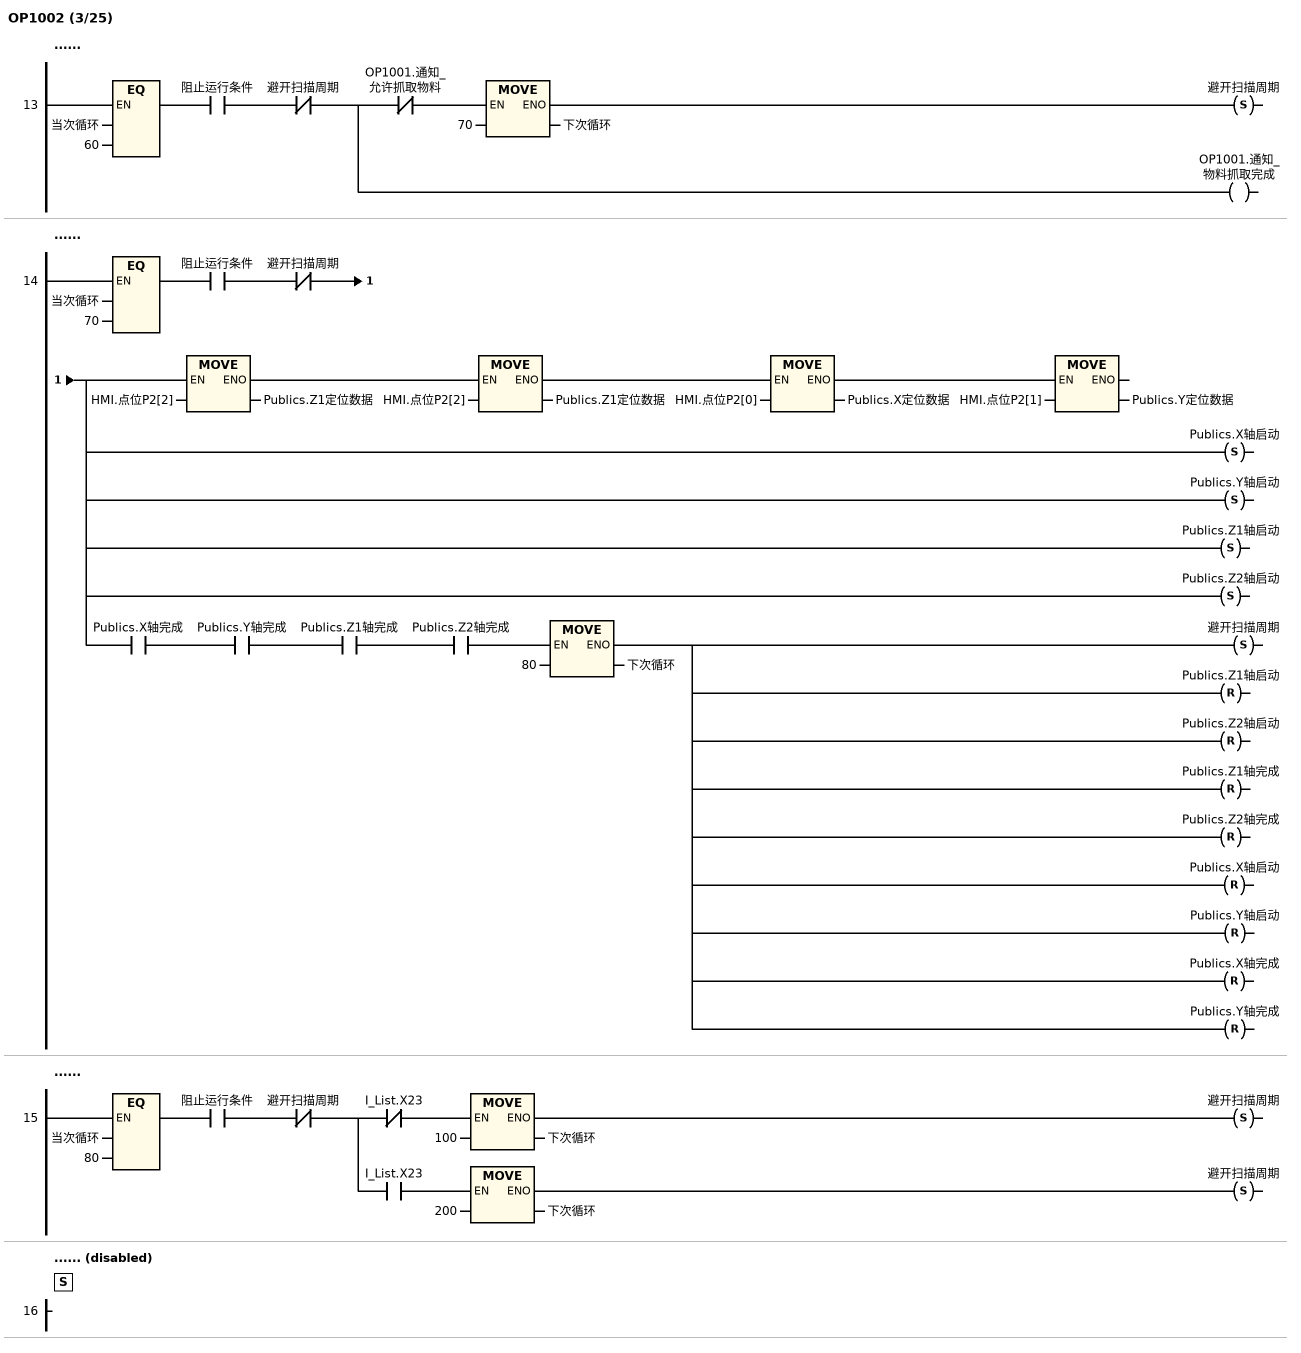
// NETWORK 13: ......
_w9 := 当次循环 = 60 AND 阻止运行条件 AND NOT 避开扫描周期;
IF _w9 AND NOT OP1001.通知_允许抓取物料 THEN 下次循环 := 70; END_IF
避开扫描周期 S= _w9 AND NOT OP1001.通知_允许抓取物料;
OP1001.通知_物料抓取完成 := _w9;

// NETWORK 14: ......
_w10 := 当次循环 = 70 AND 阻止运行条件 AND NOT 避开扫描周期;
IF _w10 THEN Publics.Z1定位数据 := HMI.点位P2[2]; END_IF
IF _w10 THEN Publics.Z1定位数据 := HMI.点位P2[2]; END_IF
IF _w10 THEN Publics.X定位数据 := HMI.点位P2[0]; END_IF
IF _w10 THEN Publics.Y定位数据 := HMI.点位P2[1]; END_IF
Publics.X轴启动 S= _w10;
Publics.Y轴启动 S= _w10;
Publics.Z1轴启动 S= _w10;
Publics.Z2轴启动 S= _w10;
IF _w10 AND Publics.X轴完成 AND Publics.Y轴完成 AND Publics.Z1轴完成 AND Publics.Z2轴完成 THEN 下次循环 := 80; END_IF
_w11 := _w10 AND Publics.X轴完成 AND Publics.Y轴完成 AND Publics.Z1轴完成 AND Publics.Z2轴完成;
避开扫描周期 S= _w11;
Publics.Z1轴启动 R= _w11;
Publics.Z2轴启动 R= _w11;
Publics.Z1轴完成 R= _w11;
Publics.Z2轴完成 R= _w11;
Publics.X轴启动 R= _w11;
Publics.Y轴启动 R= _w11;
Publics.X轴完成 R= _w11;
Publics.Y轴完成 R= _w11;

// NETWORK 15: ......
_w12 := 当次循环 = 80 AND 阻止运行条件 AND NOT 避开扫描周期;
IF _w12 AND NOT I_List.X23 THEN 下次循环 := 100; END_IF
避开扫描周期 S= _w12 AND NOT I_List.X23;
IF _w12 AND I_List.X23 THEN 下次循环 := 200; END_IF
避开扫描周期 S= _w12 AND I_List.X23;

// NETWORK 16: ...... (disabled)
// label: S

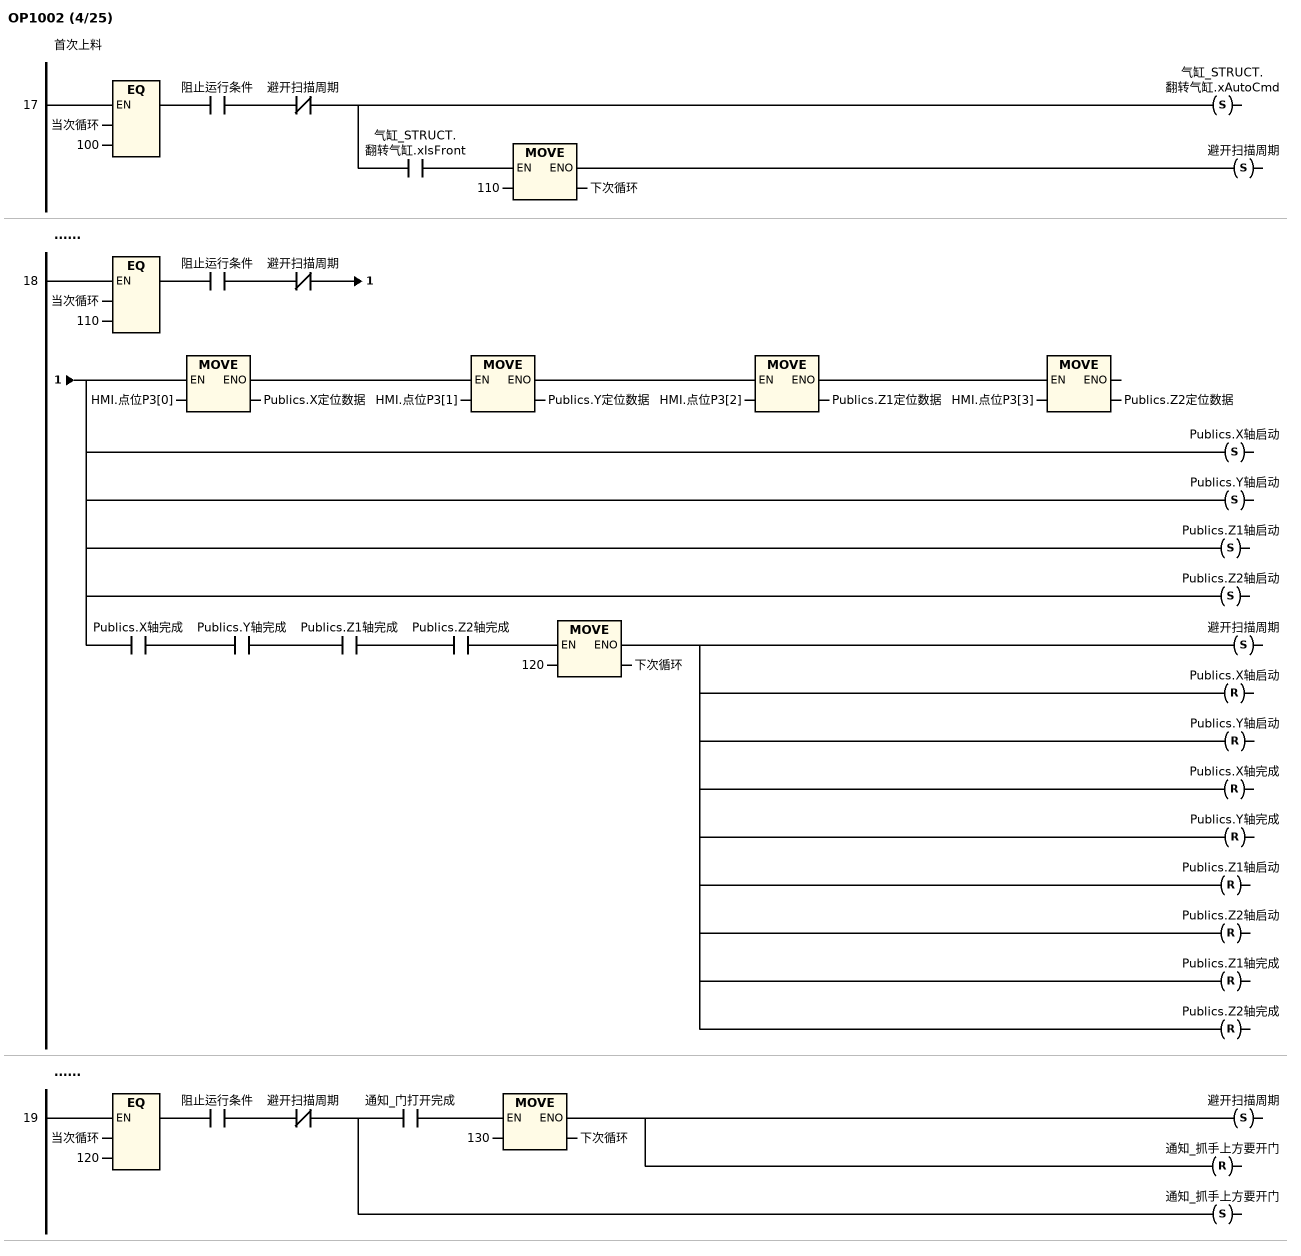
// NETWORK 17: 首次上料
_w13 := 当次循环 = 100 AND 阻止运行条件 AND NOT 避开扫描周期;
气缸_STRUCT.翻转气缸.xAutoCmd S= _w13;
IF _w13 AND 气缸_STRUCT.翻转气缸.xIsFront THEN 下次循环 := 110; END_IF
避开扫描周期 S= _w13 AND 气缸_STRUCT.翻转气缸.xIsFront;

// NETWORK 18: ......
_w14 := 当次循环 = 110 AND 阻止运行条件 AND NOT 避开扫描周期;
IF _w14 THEN Publics.X定位数据 := HMI.点位P3[0]; END_IF
IF _w14 THEN Publics.Y定位数据 := HMI.点位P3[1]; END_IF
IF _w14 THEN Publics.Z1定位数据 := HMI.点位P3[2]; END_IF
IF _w14 THEN Publics.Z2定位数据 := HMI.点位P3[3]; END_IF
Publics.X轴启动 S= _w14;
Publics.Y轴启动 S= _w14;
Publics.Z1轴启动 S= _w14;
Publics.Z2轴启动 S= _w14;
IF _w14 AND Publics.X轴完成 AND Publics.Y轴完成 AND Publics.Z1轴完成 AND Publics.Z2轴完成 THEN 下次循环 := 120; END_IF
_w15 := _w14 AND Publics.X轴完成 AND Publics.Y轴完成 AND Publics.Z1轴完成 AND Publics.Z2轴完成;
避开扫描周期 S= _w15;
Publics.X轴启动 R= _w15;
Publics.Y轴启动 R= _w15;
Publics.X轴完成 R= _w15;
Publics.Y轴完成 R= _w15;
Publics.Z1轴启动 R= _w15;
Publics.Z2轴启动 R= _w15;
Publics.Z1轴完成 R= _w15;
Publics.Z2轴完成 R= _w15;

// NETWORK 19: ......
_w16 := 当次循环 = 120 AND 阻止运行条件 AND NOT 避开扫描周期;
IF _w16 AND 通知_门打开完成 THEN 下次循环 := 130; END_IF
_w17 := _w16 AND 通知_门打开完成;
避开扫描周期 S= _w17;
通知_抓手上方要开门 R= _w17;
通知_抓手上方要开门 S= _w16;

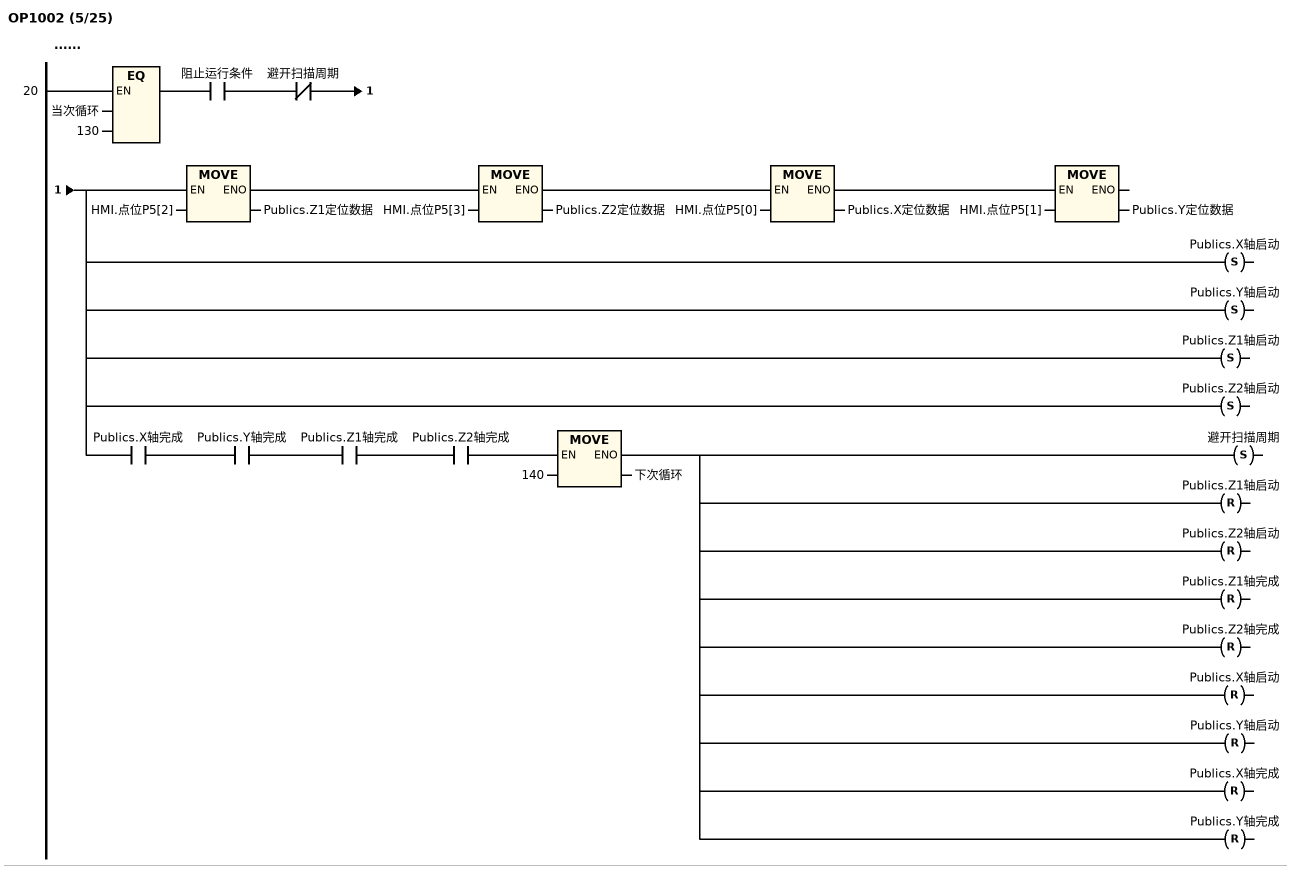
// NETWORK 20: ......
_w18 := 当次循环 = 130 AND 阻止运行条件 AND NOT 避开扫描周期;
IF _w18 THEN Publics.Z1定位数据 := HMI.点位P5[2]; END_IF
IF _w18 THEN Publics.Z2定位数据 := HMI.点位P5[3]; END_IF
IF _w18 THEN Publics.X定位数据 := HMI.点位P5[0]; END_IF
IF _w18 THEN Publics.Y定位数据 := HMI.点位P5[1]; END_IF
Publics.X轴启动 S= _w18;
Publics.Y轴启动 S= _w18;
Publics.Z1轴启动 S= _w18;
Publics.Z2轴启动 S= _w18;
IF _w18 AND Publics.X轴完成 AND Publics.Y轴完成 AND Publics.Z1轴完成 AND Publics.Z2轴完成 THEN 下次循环 := 140; END_IF
_w19 := _w18 AND Publics.X轴完成 AND Publics.Y轴完成 AND Publics.Z1轴完成 AND Publics.Z2轴完成;
避开扫描周期 S= _w19;
Publics.Z1轴启动 R= _w19;
Publics.Z2轴启动 R= _w19;
Publics.Z1轴完成 R= _w19;
Publics.Z2轴完成 R= _w19;
Publics.X轴启动 R= _w19;
Publics.Y轴启动 R= _w19;
Publics.X轴完成 R= _w19;
Publics.Y轴完成 R= _w19;

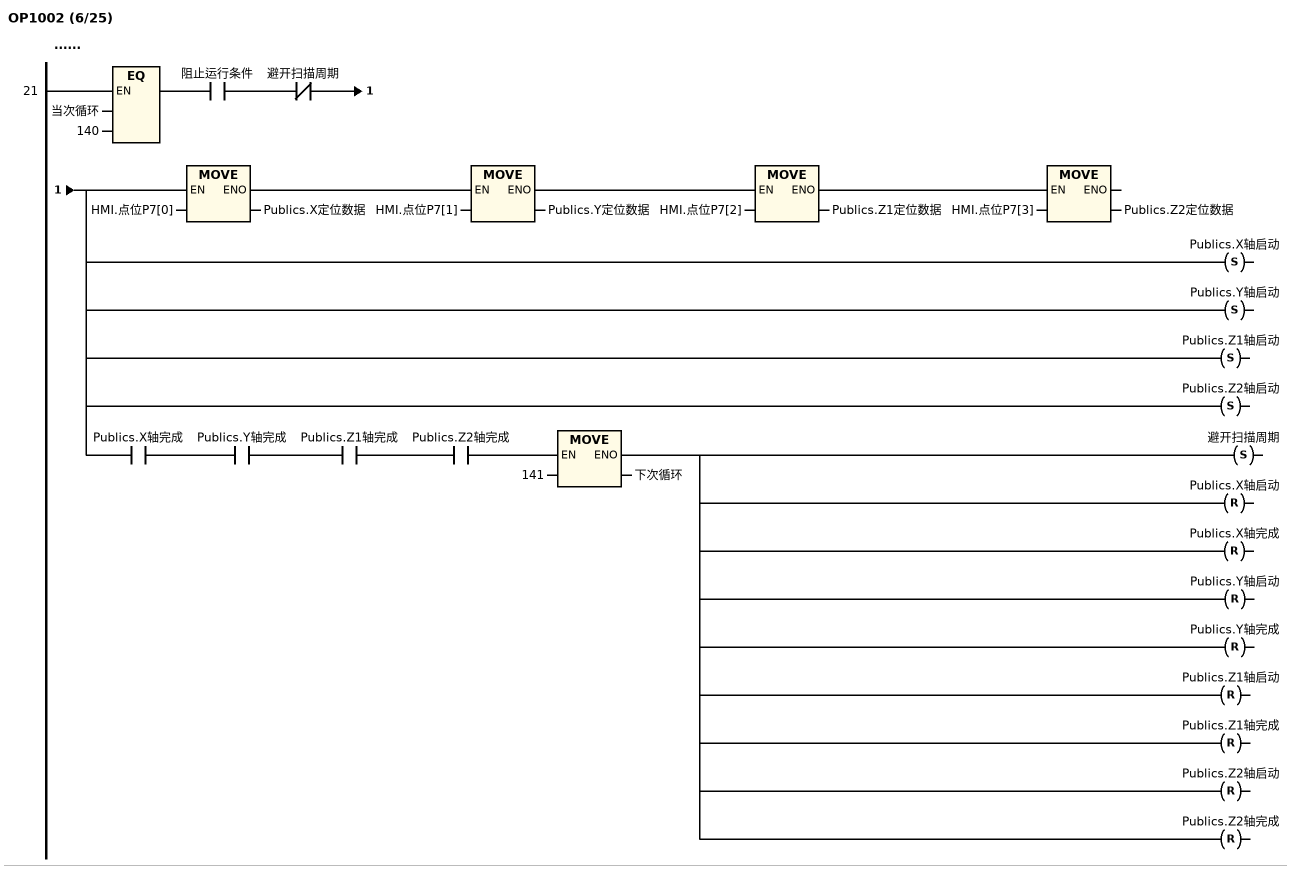
// NETWORK 21: ......
_w20 := 当次循环 = 140 AND 阻止运行条件 AND NOT 避开扫描周期;
IF _w20 THEN Publics.X定位数据 := HMI.点位P7[0]; END_IF
IF _w20 THEN Publics.Y定位数据 := HMI.点位P7[1]; END_IF
IF _w20 THEN Publics.Z1定位数据 := HMI.点位P7[2]; END_IF
IF _w20 THEN Publics.Z2定位数据 := HMI.点位P7[3]; END_IF
Publics.X轴启动 S= _w20;
Publics.Y轴启动 S= _w20;
Publics.Z1轴启动 S= _w20;
Publics.Z2轴启动 S= _w20;
IF _w20 AND Publics.X轴完成 AND Publics.Y轴完成 AND Publics.Z1轴完成 AND Publics.Z2轴完成 THEN 下次循环 := 141; END_IF
_w21 := _w20 AND Publics.X轴完成 AND Publics.Y轴完成 AND Publics.Z1轴完成 AND Publics.Z2轴完成;
避开扫描周期 S= _w21;
Publics.X轴启动 R= _w21;
Publics.X轴完成 R= _w21;
Publics.Y轴启动 R= _w21;
Publics.Y轴完成 R= _w21;
Publics.Z1轴启动 R= _w21;
Publics.Z1轴完成 R= _w21;
Publics.Z2轴启动 R= _w21;
Publics.Z2轴完成 R= _w21;

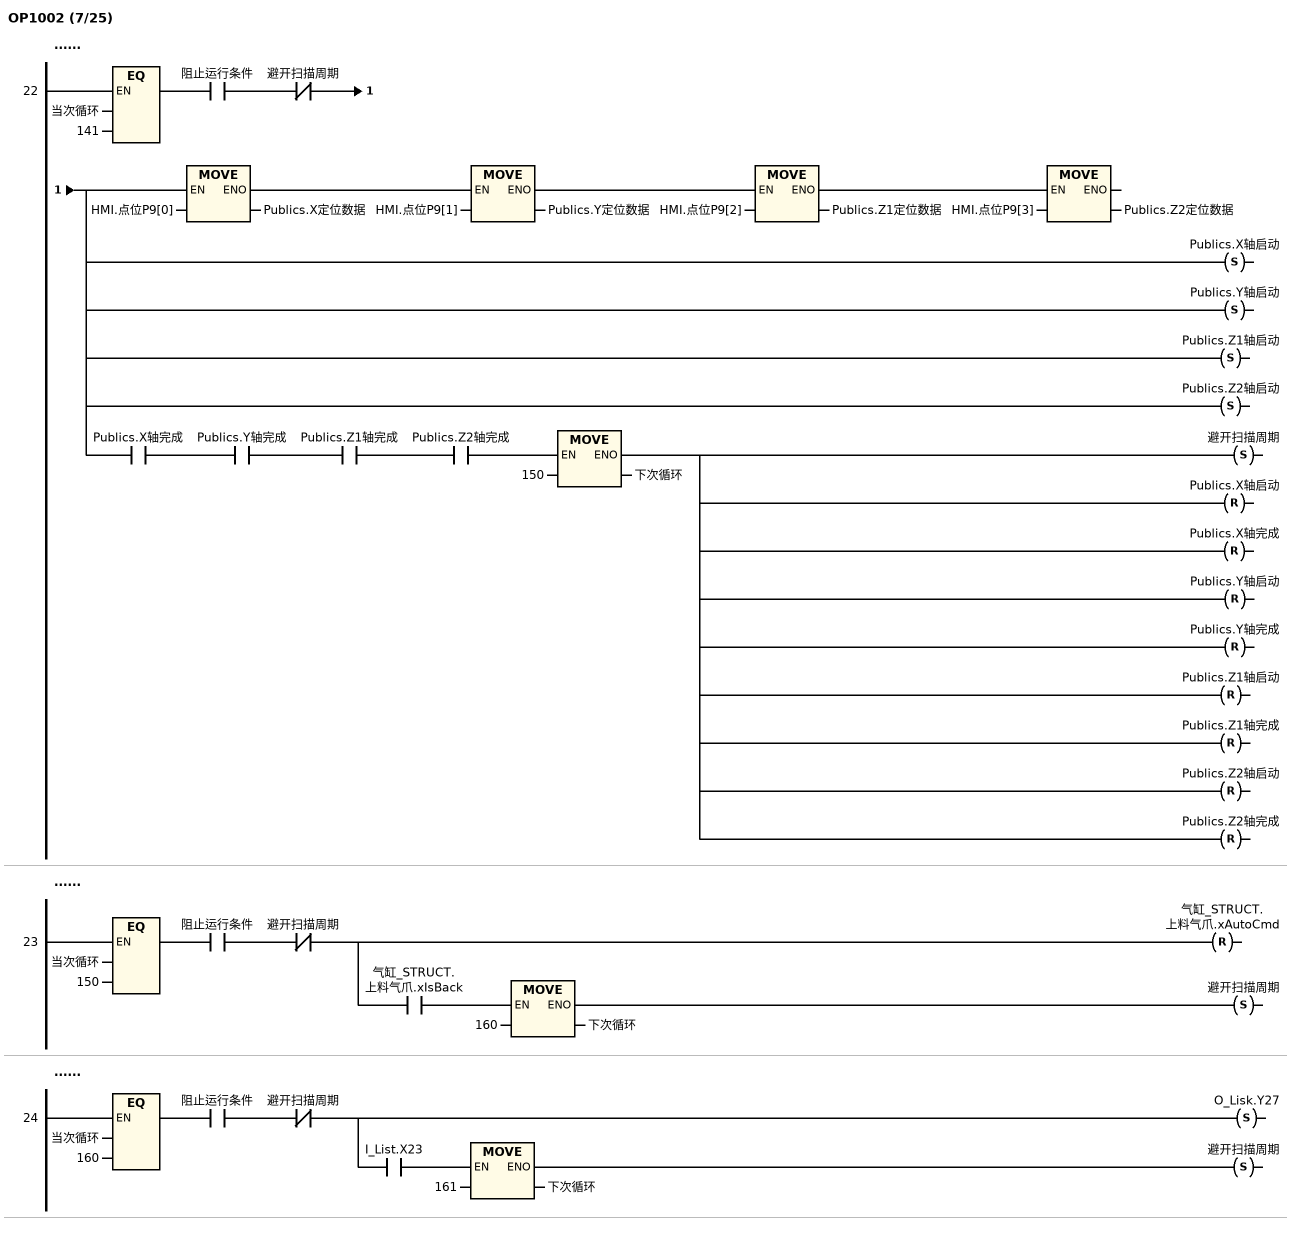
// NETWORK 22: ......
_w22 := 当次循环 = 141 AND 阻止运行条件 AND NOT 避开扫描周期;
IF _w22 THEN Publics.X定位数据 := HMI.点位P9[0]; END_IF
IF _w22 THEN Publics.Y定位数据 := HMI.点位P9[1]; END_IF
IF _w22 THEN Publics.Z1定位数据 := HMI.点位P9[2]; END_IF
IF _w22 THEN Publics.Z2定位数据 := HMI.点位P9[3]; END_IF
Publics.X轴启动 S= _w22;
Publics.Y轴启动 S= _w22;
Publics.Z1轴启动 S= _w22;
Publics.Z2轴启动 S= _w22;
IF _w22 AND Publics.X轴完成 AND Publics.Y轴完成 AND Publics.Z1轴完成 AND Publics.Z2轴完成 THEN 下次循环 := 150; END_IF
_w23 := _w22 AND Publics.X轴完成 AND Publics.Y轴完成 AND Publics.Z1轴完成 AND Publics.Z2轴完成;
避开扫描周期 S= _w23;
Publics.X轴启动 R= _w23;
Publics.X轴完成 R= _w23;
Publics.Y轴启动 R= _w23;
Publics.Y轴完成 R= _w23;
Publics.Z1轴启动 R= _w23;
Publics.Z1轴完成 R= _w23;
Publics.Z2轴启动 R= _w23;
Publics.Z2轴完成 R= _w23;

// NETWORK 23: ......
_w24 := 当次循环 = 150 AND 阻止运行条件 AND NOT 避开扫描周期;
气缸_STRUCT.上料气爪.xAutoCmd R= _w24;
IF _w24 AND 气缸_STRUCT.上料气爪.xIsBack THEN 下次循环 := 160; END_IF
避开扫描周期 S= _w24 AND 气缸_STRUCT.上料气爪.xIsBack;

// NETWORK 24: ......
_w25 := 当次循环 = 160 AND 阻止运行条件 AND NOT 避开扫描周期;
O_Lisk.Y27 S= _w25;
IF _w25 AND I_List.X23 THEN 下次循环 := 161; END_IF
避开扫描周期 S= _w25 AND I_List.X23;

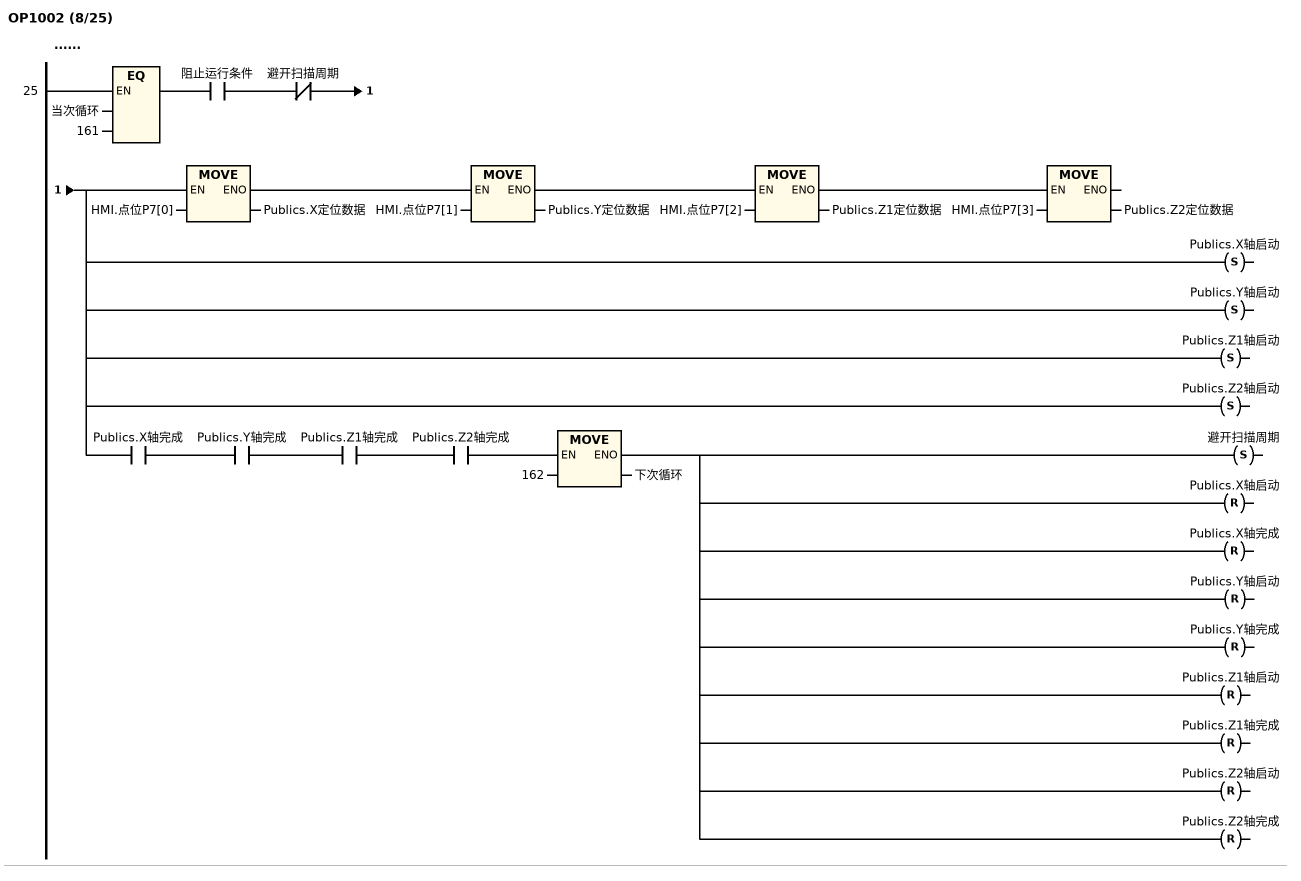
// NETWORK 25: ......
_w26 := 当次循环 = 161 AND 阻止运行条件 AND NOT 避开扫描周期;
IF _w26 THEN Publics.X定位数据 := HMI.点位P7[0]; END_IF
IF _w26 THEN Publics.Y定位数据 := HMI.点位P7[1]; END_IF
IF _w26 THEN Publics.Z1定位数据 := HMI.点位P7[2]; END_IF
IF _w26 THEN Publics.Z2定位数据 := HMI.点位P7[3]; END_IF
Publics.X轴启动 S= _w26;
Publics.Y轴启动 S= _w26;
Publics.Z1轴启动 S= _w26;
Publics.Z2轴启动 S= _w26;
IF _w26 AND Publics.X轴完成 AND Publics.Y轴完成 AND Publics.Z1轴完成 AND Publics.Z2轴完成 THEN 下次循环 := 162; END_IF
_w27 := _w26 AND Publics.X轴完成 AND Publics.Y轴完成 AND Publics.Z1轴完成 AND Publics.Z2轴完成;
避开扫描周期 S= _w27;
Publics.X轴启动 R= _w27;
Publics.X轴完成 R= _w27;
Publics.Y轴启动 R= _w27;
Publics.Y轴完成 R= _w27;
Publics.Z1轴启动 R= _w27;
Publics.Z1轴完成 R= _w27;
Publics.Z2轴启动 R= _w27;
Publics.Z2轴完成 R= _w27;

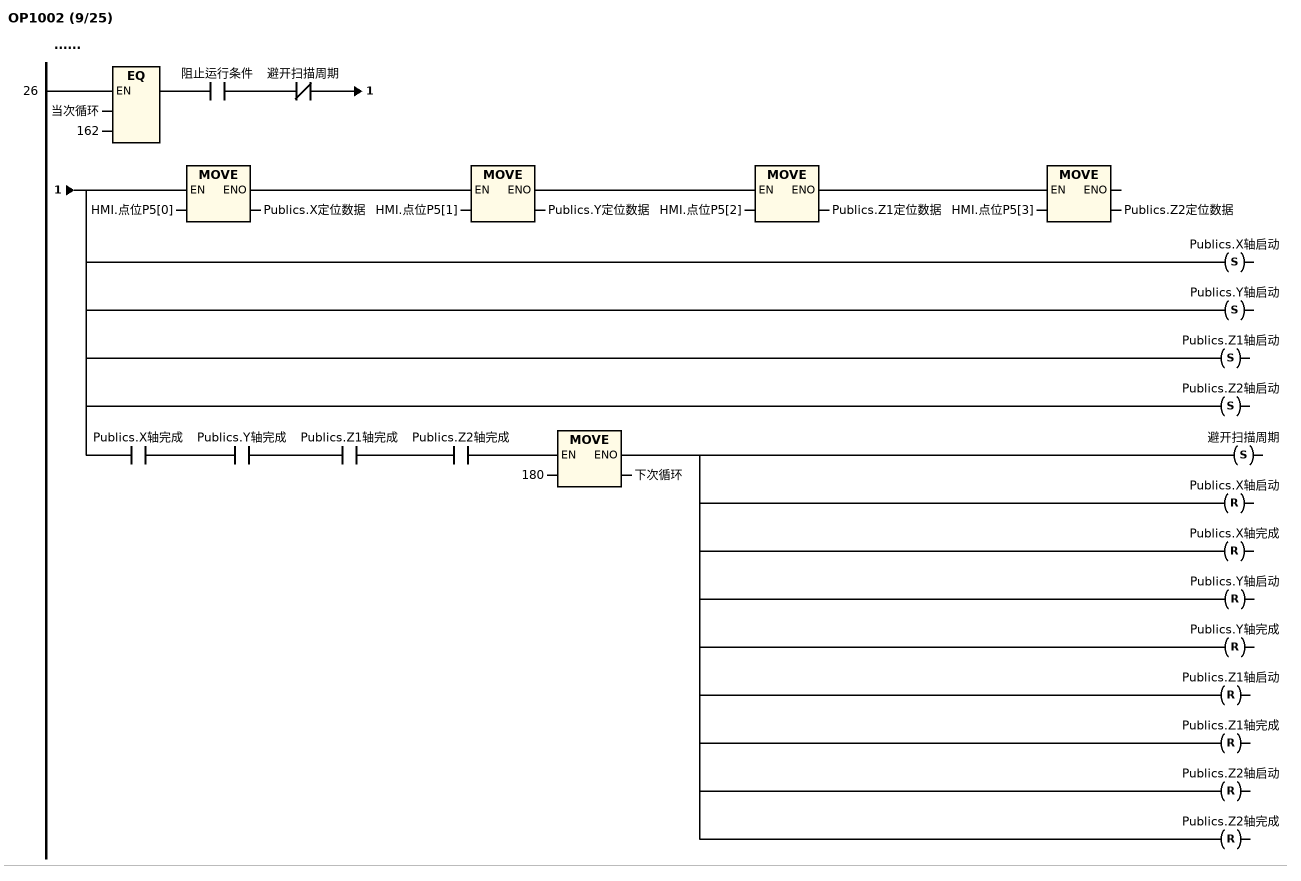
// NETWORK 26: ......
_w28 := 当次循环 = 162 AND 阻止运行条件 AND NOT 避开扫描周期;
IF _w28 THEN Publics.X定位数据 := HMI.点位P5[0]; END_IF
IF _w28 THEN Publics.Y定位数据 := HMI.点位P5[1]; END_IF
IF _w28 THEN Publics.Z1定位数据 := HMI.点位P5[2]; END_IF
IF _w28 THEN Publics.Z2定位数据 := HMI.点位P5[3]; END_IF
Publics.X轴启动 S= _w28;
Publics.Y轴启动 S= _w28;
Publics.Z1轴启动 S= _w28;
Publics.Z2轴启动 S= _w28;
IF _w28 AND Publics.X轴完成 AND Publics.Y轴完成 AND Publics.Z1轴完成 AND Publics.Z2轴完成 THEN 下次循环 := 180; END_IF
_w29 := _w28 AND Publics.X轴完成 AND Publics.Y轴完成 AND Publics.Z1轴完成 AND Publics.Z2轴完成;
避开扫描周期 S= _w29;
Publics.X轴启动 R= _w29;
Publics.X轴完成 R= _w29;
Publics.Y轴启动 R= _w29;
Publics.Y轴完成 R= _w29;
Publics.Z1轴启动 R= _w29;
Publics.Z1轴完成 R= _w29;
Publics.Z2轴启动 R= _w29;
Publics.Z2轴完成 R= _w29;

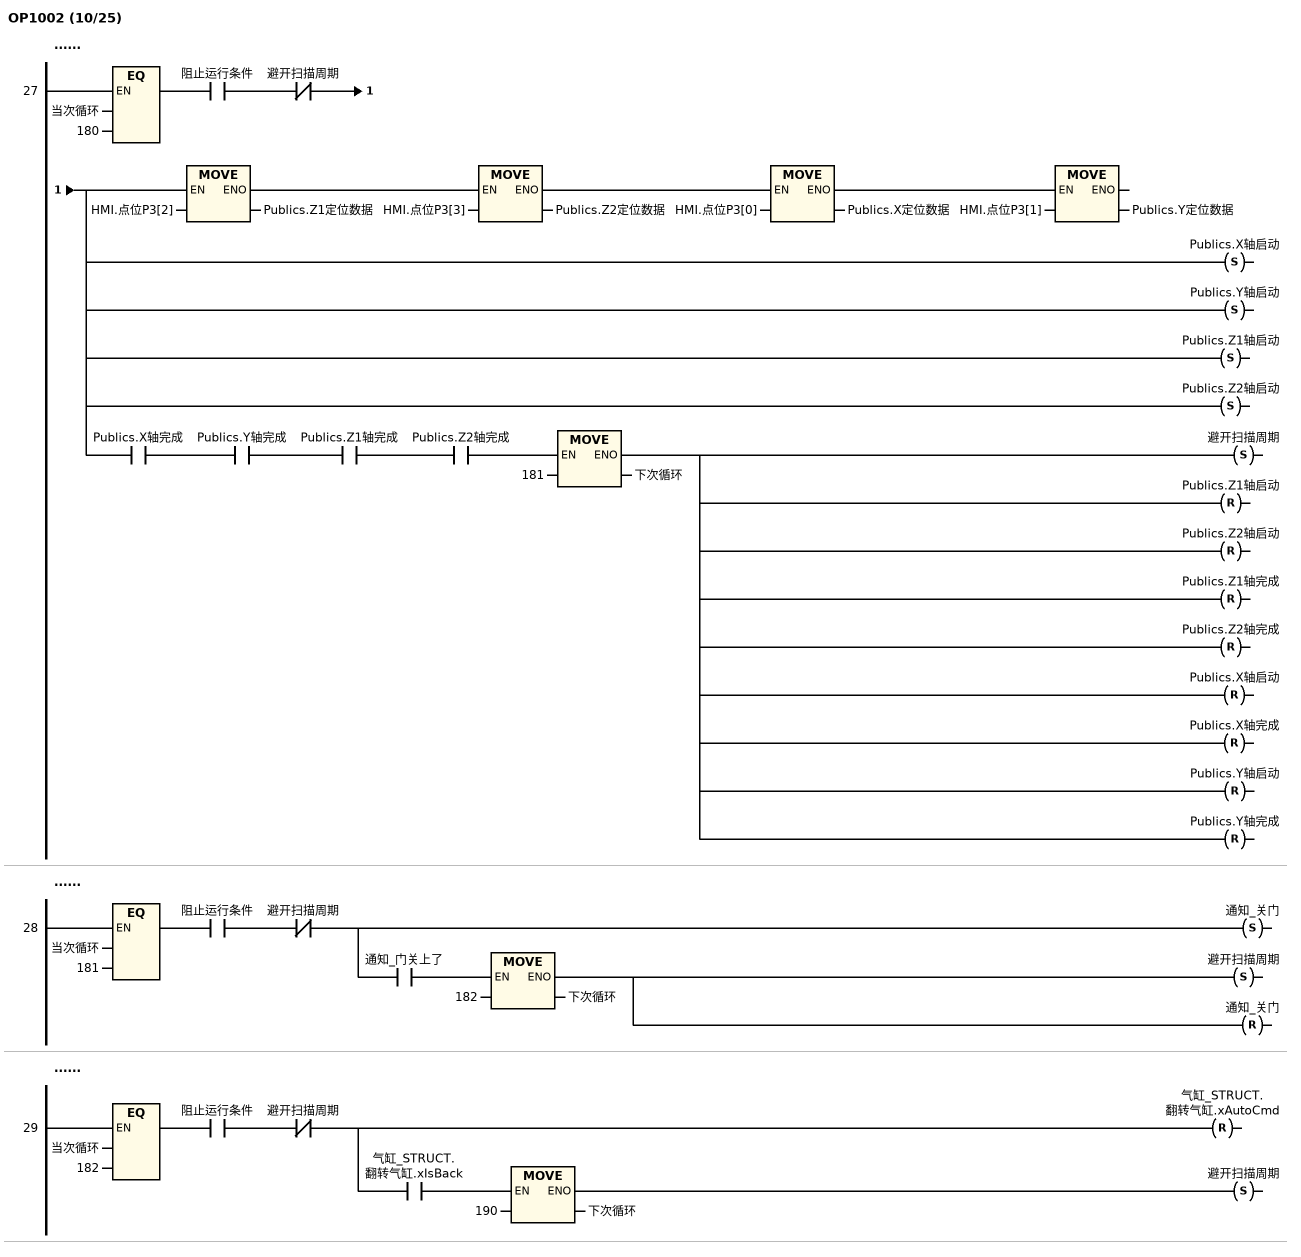
// NETWORK 27: ......
_w30 := 当次循环 = 180 AND 阻止运行条件 AND NOT 避开扫描周期;
IF _w30 THEN Publics.Z1定位数据 := HMI.点位P3[2]; END_IF
IF _w30 THEN Publics.Z2定位数据 := HMI.点位P3[3]; END_IF
IF _w30 THEN Publics.X定位数据 := HMI.点位P3[0]; END_IF
IF _w30 THEN Publics.Y定位数据 := HMI.点位P3[1]; END_IF
Publics.X轴启动 S= _w30;
Publics.Y轴启动 S= _w30;
Publics.Z1轴启动 S= _w30;
Publics.Z2轴启动 S= _w30;
IF _w30 AND Publics.X轴完成 AND Publics.Y轴完成 AND Publics.Z1轴完成 AND Publics.Z2轴完成 THEN 下次循环 := 181; END_IF
_w31 := _w30 AND Publics.X轴完成 AND Publics.Y轴完成 AND Publics.Z1轴完成 AND Publics.Z2轴完成;
避开扫描周期 S= _w31;
Publics.Z1轴启动 R= _w31;
Publics.Z2轴启动 R= _w31;
Publics.Z1轴完成 R= _w31;
Publics.Z2轴完成 R= _w31;
Publics.X轴启动 R= _w31;
Publics.X轴完成 R= _w31;
Publics.Y轴启动 R= _w31;
Publics.Y轴完成 R= _w31;

// NETWORK 28: ......
_w32 := 当次循环 = 181 AND 阻止运行条件 AND NOT 避开扫描周期;
通知_关门 S= _w32;
IF _w32 AND 通知_门关上了 THEN 下次循环 := 182; END_IF
_w33 := _w32 AND 通知_门关上了;
避开扫描周期 S= _w33;
通知_关门 R= _w33;

// NETWORK 29: ......
_w34 := 当次循环 = 182 AND 阻止运行条件 AND NOT 避开扫描周期;
气缸_STRUCT.翻转气缸.xAutoCmd R= _w34;
IF _w34 AND 气缸_STRUCT.翻转气缸.xIsBack THEN 下次循环 := 190; END_IF
避开扫描周期 S= _w34 AND 气缸_STRUCT.翻转气缸.xIsBack;

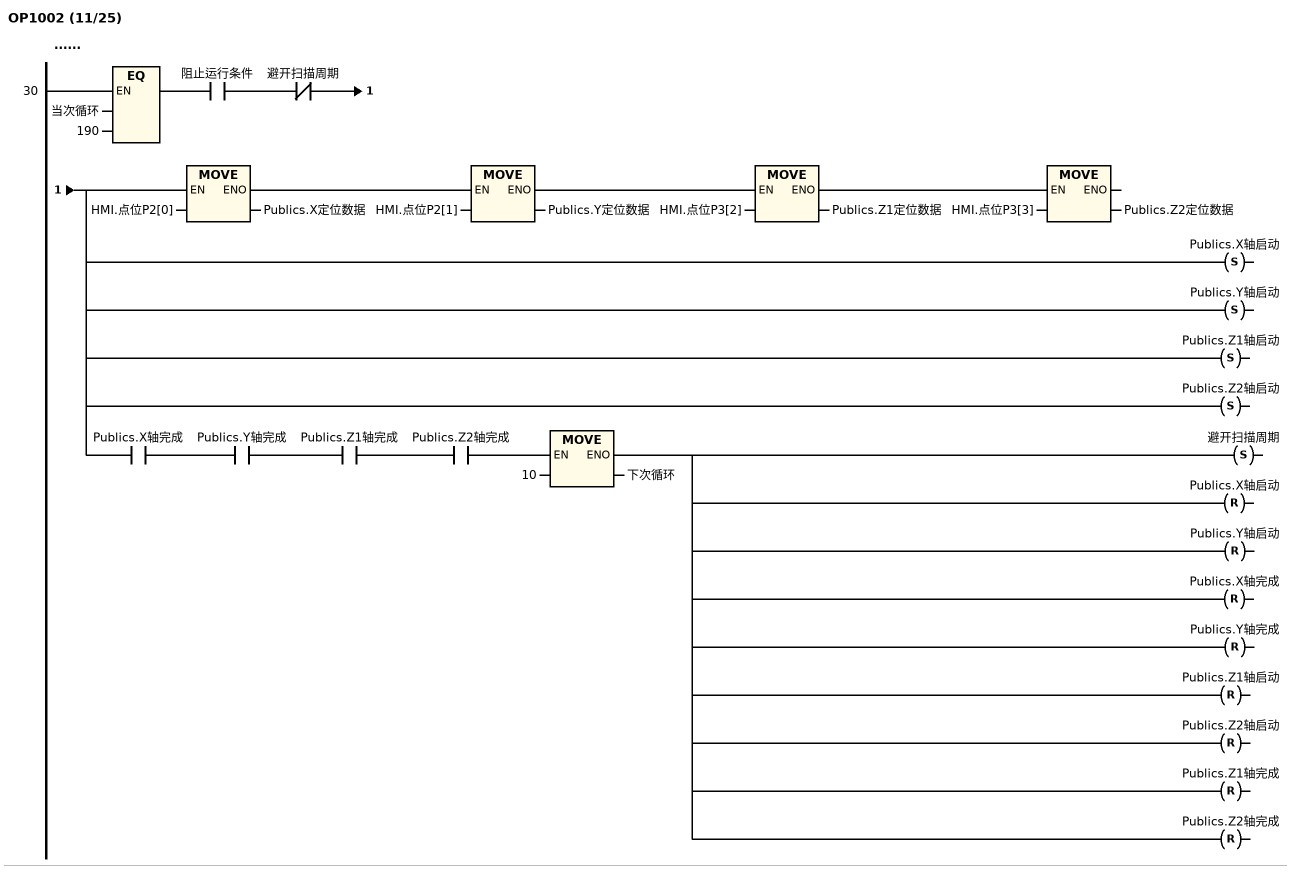
// NETWORK 30: ......
_w35 := 当次循环 = 190 AND 阻止运行条件 AND NOT 避开扫描周期;
IF _w35 THEN Publics.X定位数据 := HMI.点位P2[0]; END_IF
IF _w35 THEN Publics.Y定位数据 := HMI.点位P2[1]; END_IF
IF _w35 THEN Publics.Z1定位数据 := HMI.点位P3[2]; END_IF
IF _w35 THEN Publics.Z2定位数据 := HMI.点位P3[3]; END_IF
Publics.X轴启动 S= _w35;
Publics.Y轴启动 S= _w35;
Publics.Z1轴启动 S= _w35;
Publics.Z2轴启动 S= _w35;
IF _w35 AND Publics.X轴完成 AND Publics.Y轴完成 AND Publics.Z1轴完成 AND Publics.Z2轴完成 THEN 下次循环 := 10; END_IF
_w36 := _w35 AND Publics.X轴完成 AND Publics.Y轴完成 AND Publics.Z1轴完成 AND Publics.Z2轴完成;
避开扫描周期 S= _w36;
Publics.X轴启动 R= _w36;
Publics.Y轴启动 R= _w36;
Publics.X轴完成 R= _w36;
Publics.Y轴完成 R= _w36;
Publics.Z1轴启动 R= _w36;
Publics.Z2轴启动 R= _w36;
Publics.Z1轴完成 R= _w36;
Publics.Z2轴完成 R= _w36;

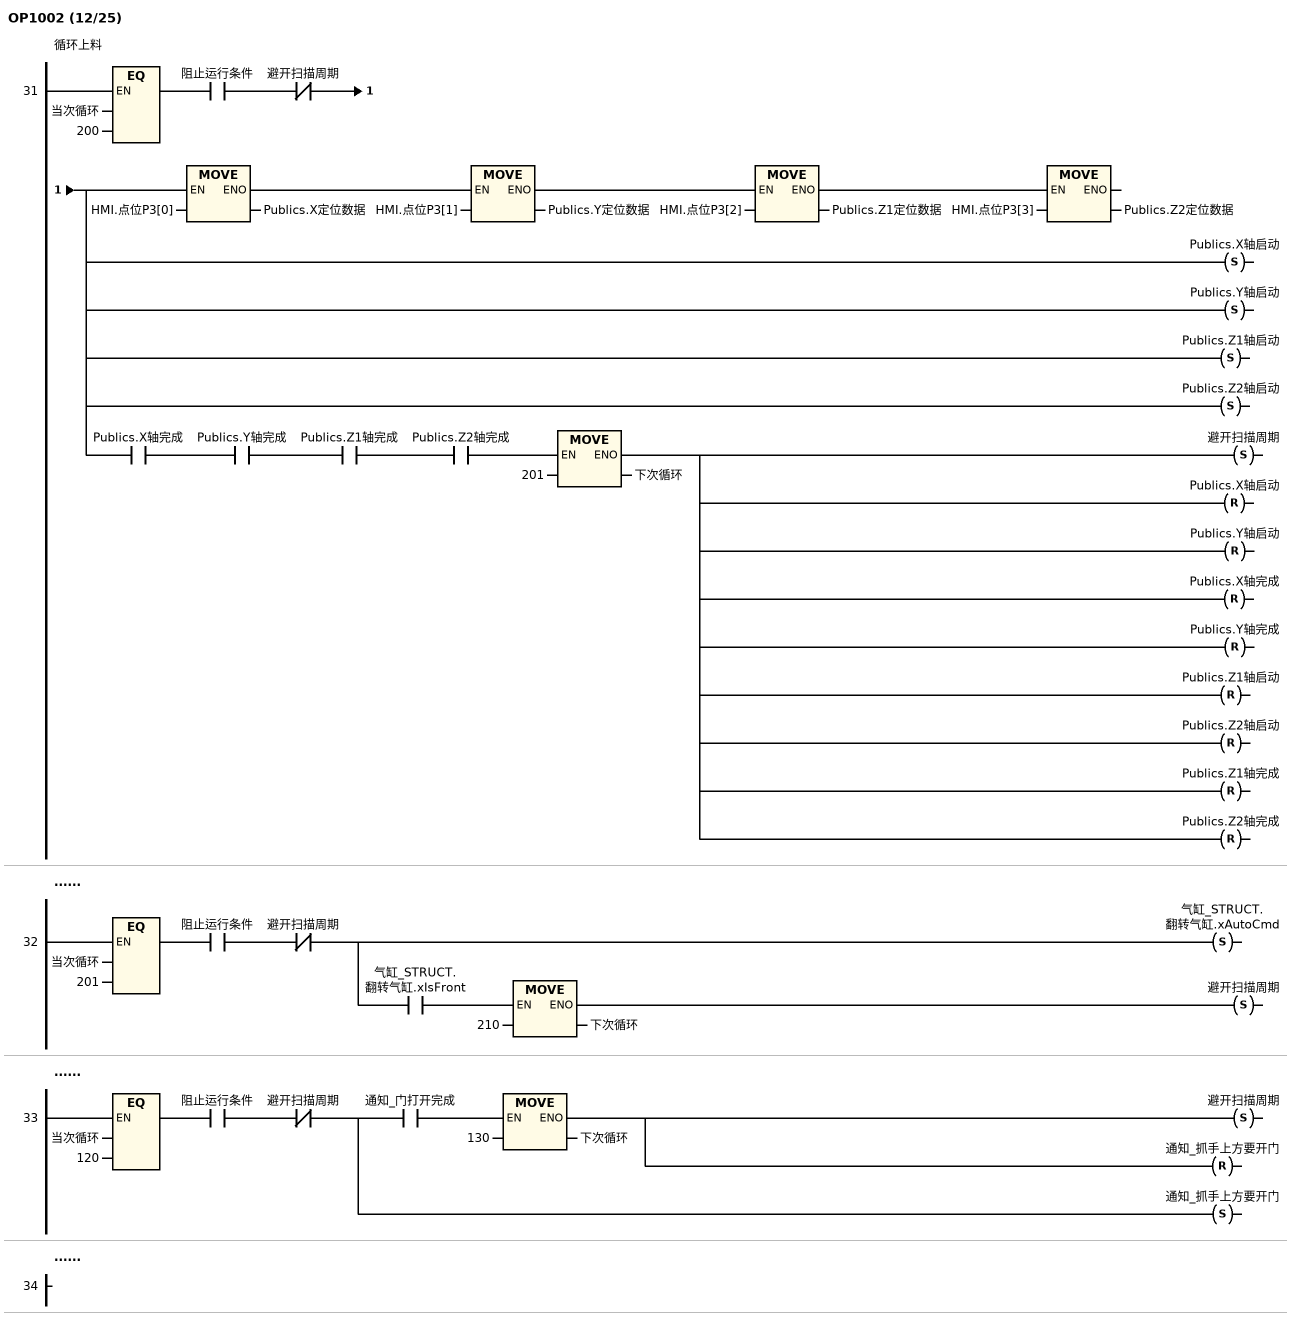
// NETWORK 31: 循环上料
_w37 := 当次循环 = 200 AND 阻止运行条件 AND NOT 避开扫描周期;
IF _w37 THEN Publics.X定位数据 := HMI.点位P3[0]; END_IF
IF _w37 THEN Publics.Y定位数据 := HMI.点位P3[1]; END_IF
IF _w37 THEN Publics.Z1定位数据 := HMI.点位P3[2]; END_IF
IF _w37 THEN Publics.Z2定位数据 := HMI.点位P3[3]; END_IF
Publics.X轴启动 S= _w37;
Publics.Y轴启动 S= _w37;
Publics.Z1轴启动 S= _w37;
Publics.Z2轴启动 S= _w37;
IF _w37 AND Publics.X轴完成 AND Publics.Y轴完成 AND Publics.Z1轴完成 AND Publics.Z2轴完成 THEN 下次循环 := 201; END_IF
_w38 := _w37 AND Publics.X轴完成 AND Publics.Y轴完成 AND Publics.Z1轴完成 AND Publics.Z2轴完成;
避开扫描周期 S= _w38;
Publics.X轴启动 R= _w38;
Publics.Y轴启动 R= _w38;
Publics.X轴完成 R= _w38;
Publics.Y轴完成 R= _w38;
Publics.Z1轴启动 R= _w38;
Publics.Z2轴启动 R= _w38;
Publics.Z1轴完成 R= _w38;
Publics.Z2轴完成 R= _w38;

// NETWORK 32: ......
_w39 := 当次循环 = 201 AND 阻止运行条件 AND NOT 避开扫描周期;
气缸_STRUCT.翻转气缸.xAutoCmd S= _w39;
IF _w39 AND 气缸_STRUCT.翻转气缸.xIsFront THEN 下次循环 := 210; END_IF
避开扫描周期 S= _w39 AND 气缸_STRUCT.翻转气缸.xIsFront;

// NETWORK 33: ......
_w40 := 当次循环 = 120 AND 阻止运行条件 AND NOT 避开扫描周期;
IF _w40 AND 通知_门打开完成 THEN 下次循环 := 130; END_IF
_w41 := _w40 AND 通知_门打开完成;
避开扫描周期 S= _w41;
通知_抓手上方要开门 R= _w41;
通知_抓手上方要开门 S= _w40;

// NETWORK 34: ......

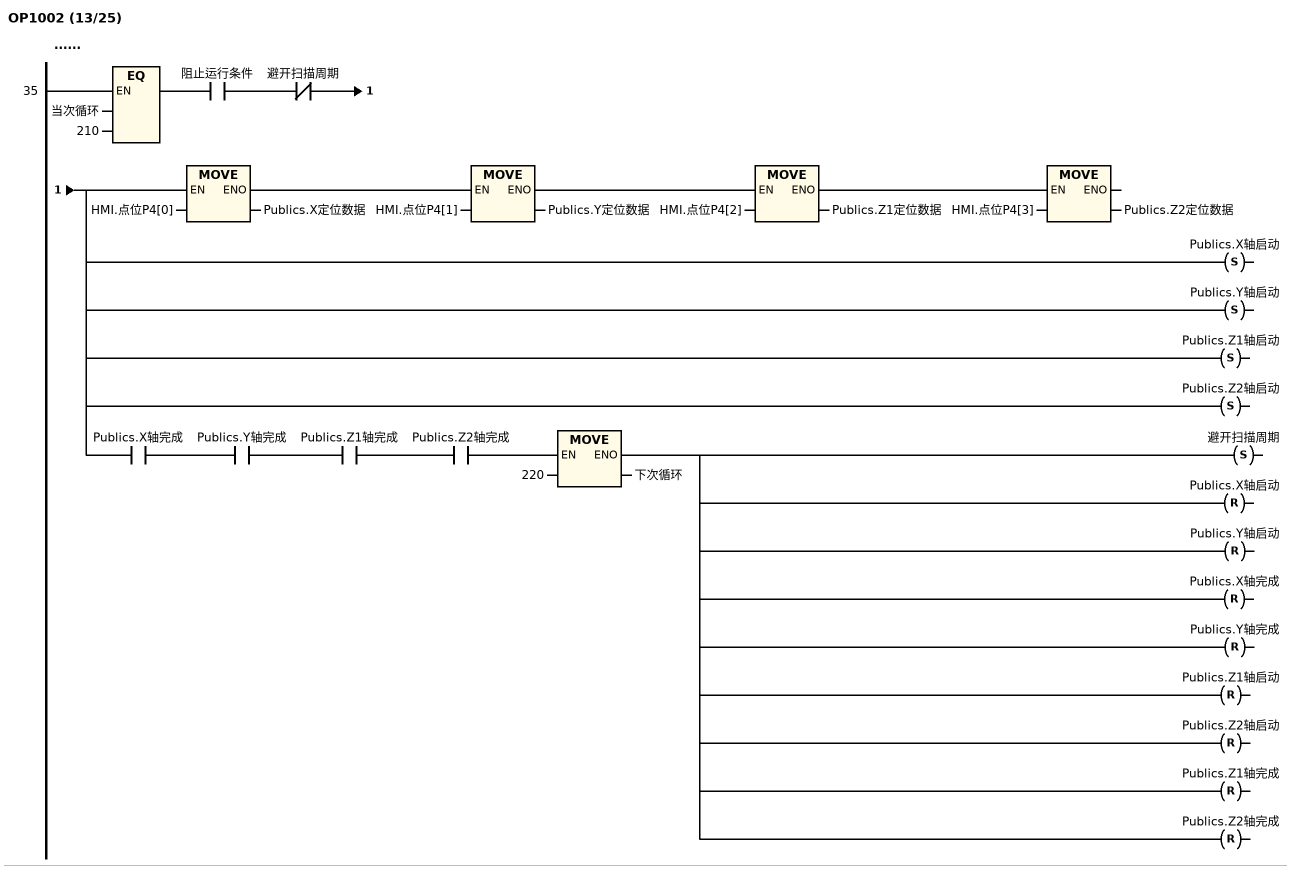
// NETWORK 35: ......
_w42 := 当次循环 = 210 AND 阻止运行条件 AND NOT 避开扫描周期;
IF _w42 THEN Publics.X定位数据 := HMI.点位P4[0]; END_IF
IF _w42 THEN Publics.Y定位数据 := HMI.点位P4[1]; END_IF
IF _w42 THEN Publics.Z1定位数据 := HMI.点位P4[2]; END_IF
IF _w42 THEN Publics.Z2定位数据 := HMI.点位P4[3]; END_IF
Publics.X轴启动 S= _w42;
Publics.Y轴启动 S= _w42;
Publics.Z1轴启动 S= _w42;
Publics.Z2轴启动 S= _w42;
IF _w42 AND Publics.X轴完成 AND Publics.Y轴完成 AND Publics.Z1轴完成 AND Publics.Z2轴完成 THEN 下次循环 := 220; END_IF
_w43 := _w42 AND Publics.X轴完成 AND Publics.Y轴完成 AND Publics.Z1轴完成 AND Publics.Z2轴完成;
避开扫描周期 S= _w43;
Publics.X轴启动 R= _w43;
Publics.Y轴启动 R= _w43;
Publics.X轴完成 R= _w43;
Publics.Y轴完成 R= _w43;
Publics.Z1轴启动 R= _w43;
Publics.Z2轴启动 R= _w43;
Publics.Z1轴完成 R= _w43;
Publics.Z2轴完成 R= _w43;

